Yaskawa INFORM job: X2_38-47,64(1)(90,180).JBI

/JOB
//NAME X2_38-47,64(1)(90,180)
//POS
///NPOS 755,755,755,26,0,0
///TOOL 0
///POSTYPE PULSE
///PULSE
C00000=-10776,-116726,-133110,1428,79202,268
C00001=-121301,-101656,-130574,-15140,106953,-26685
C00002=-120740,-100574,-124017,-14929,103680,-26084
C00003=-120691,-100743,-123189,-14892,103111,-25997
C00004=-120691,-101012,-123023,-14875,102879,-25968
C00005=-120694,-100727,-123199,-14892,103125,-25999
C00006=-120263,-93974,-120700,-15099,105066,-26103
C00007=-120694,-100727,-123199,-14892,103125,-25999
C00008=-121303,-103883,-129892,-15002,105440,-26491
C00009=-121309,-101301,-130428,-15148,107041,-26699
C00010=-120755,-99767,-124232,-14968,104207,-26155
C00011=-120700,-99774,-123449,-14938,103747,-26079
C00012=-120700,-100712,-122892,-14879,102948,-25979
C00013=-120685,-100384,-123078,-14901,103225,-26009
C00014=-120255,-93653,-120581,-15108,105156,-26112
C00015=-120685,-100384,-123078,-14901,103225,-26009
C00016=-121293,-103472,-129753,-15014,105563,-26504
C00017=-114791,-117911,-130965,-19588,74628,-29967
C00018=-114769,-122713,-124135,-20312,68344,-28880
C00019=-114477,-110584,-116158,-20272,69659,-29005
C00020=-114421,-108517,-114081,-20323,69469,-28951
C00021=-114421,-108669,-113508,-20377,69064,-28879
C00022=-114502,-108614,-114130,-20291,69431,-28974
C00023=-116741,-105993,-113204,-19215,69642,-29832
C00024=-114502,-108614,-114130,-20291,69431,-28974
C00025=-119599,-132627,-121815,-19129,61042,-29452
C00026=-135151,-106131,-113172,-10502,66286,-36044
C00027=-134382,-104032,-112419,-10838,66989,-35834
C00028=-133562,-101757,-111587,-11194,67742,-35614
C00029=-135151,-106131,-113172,-10502,66286,-36044
C00030=-114538,-130880,-126635,-20790,65904,-28347
C00031=-100256,-119338,-132400,-19781,92736,17009
C00032=-115252,-134637,-128783,-15911,82002,19716
C00033=-118597,-124593,-122817,-15129,82811,18454
C00034=-119849,-120977,-120499,-14834,83003,18000
C00035=-119848,-121103,-118880,-14863,81976,18124
C00036=-119849,-120977,-120499,-14834,83003,18000
C00037=-134184,-142802,-124917,-2858,68148,11180
C00038=-133176,-135816,-122960,-3144,70568,11480
C00039=-134184,-142802,-124917,-2858,68148,11180
C00040=-110326,-92448,-108322,-23569,98205,21456
C00041=-112623,-92143,-108201,-23254,97666,20755
C00042=-110326,-92448,-108322,-23569,98205,21456
C00043=-105090,-96290,-113946,-24376,100996,22735
C00044=-105112,-88407,-119445,-25319,107768,21250
C00045=-126458,-130213,-127441,18734,86324,-24062
C00046=-122565,-122494,-122126,18005,86127,-22734
C00047=-121090,-119592,-120022,17718,85999,-22241
C00048=-121089,-119765,-118419,17734,84972,-22390
C00049=-121090,-119592,-120022,17718,85999,-22241
C00050=-121090,-119716,-118696,17731,85160,-22363
C00051=-120619,-113401,-116618,17615,86937,-21943
C00052=-121090,-119716,-118696,17731,85160,-22363
C00053=-120691,-116357,-117549,17638,86049,-22096
C00054=-118089,-117386,-117887,17123,85200,-21315
C00055=-120691,-116357,-117549,17638,86049,-22096
C00056=-125936,-126318,-124843,18636,86589,-23840
C00057=-125953,-122568,-132013,18690,92614,-22924
C00058=-117644,-124381,-130105,-6983,115370,67992
C00059=-119593,-136528,-130318,-6950,109138,67660
C00060=-120425,-140611,-129416,-6959,106433,67520
C00061=-120425,-140322,-128375,-6938,105944,67549
C00062=-120287,-139878,-129033,-6943,106584,67561
C00063=-121808,-147552,-131144,-7070,103828,67181
C00064=-120287,-139878,-129033,-6943,106584,67561
C00065=-117523,-124132,-129146,-6933,114921,68065
C00066=-117634,-108923,-132591,-7489,118176,67765
C00067=-119077,-97405,-129626,-2848,111310,9091
C00068=-112934,-122170,-124968,-9693,82630,11419
C00069=-114889,-112052,-118675,-9157,83718,10686
C00070=-115614,-108714,-115508,-8968,83408,10468
C00071=-115614,-108962,-114752,-8976,82823,10510
C00072=-115614,-108688,-115602,-8966,83479,10463
C00073=-130338,-117040,-117457,5173,77211,4432
C00074=-129550,-114521,-116623,4914,77941,4728
C00075=-131152,-119600,-118288,5441,76463,4123
C00076=-115450,-106601,-114144,-9007,83670,10503
C00077=-117654,-103921,-113183,-8408,84218,9737
C00078=-115450,-106601,-114144,-9007,83670,10503
C00079=-112794,-119726,-122752,-9732,82540,11472
C00080=-112816,-114614,-129461,-9677,89201,10949
C00081=-124267,-125778,-125536,12618,81617,-14637
C00082=-121749,-115664,-119377,11934,82621,-13684
C00083=-120813,-112238,-116231,11692,82317,-13397
C00084=-120812,-112414,-115451,11705,81758,-13450
C00085=-120848,-112349,-116241,11703,82272,-13413
C00086=-119586,-107060,-114409,11339,83657,-12862
C00087=-120848,-112349,-116241,11703,82272,-13413
C00088=-124307,-126037,-124767,12644,81031,-14711
C00089=-124281,-122814,-131176,12539,86499,-14147
C00090=-130647,-155525,-127944,40400,54320,-55258
C00091=-124412,-146323,-123540,36852,53123,-52512
C00092=-122059,-142698,-121760,35413,52755,-51453
C00093=-119008,-142706,-121763,33902,51510,-50382
C00094=-122059,-142698,-121760,35413,52755,-51453
C00095=-119813,-142714,-121776,34308,51836,-50667
C00096=-119829,-137326,-119074,33845,52767,-50322
C00097=-119813,-142714,-121776,34308,51836,-50667
C00098=-119893,-119020,-120433,30427,61542,-47434
C00099=-120958,-113296,-116932,30756,62602,-47571
C00100=-120971,-118070,-117370,31352,60722,-48150
C00101=-120958,-113296,-116932,30756,62602,-47571
C00102=-130647,-155525,-127944,40400,54320,-55258
C00103=-121972,-140000,-127461,3525,22047,-40740
C00104=-114503,-126631,-127045,-28228,88345,-28238
C00105=-115418,-120062,-121213,-28067,87856,-28460
C00106=-115767,-117777,-118144,-28010,87108,-28410
C00107=-115767,-117863,-117333,-28016,86625,-28294
C00108=-115798,-117876,-117463,-28010,86680,-28319
C00109=-115506,-111666,-115391,-28051,88476,-28642
C00110=-115798,-117876,-117463,-28010,86680,-28319
C00111=-114535,-126949,-125608,-28226,87406,-28022
C00112=-81132,-132100,-132064,-22325,96940,-18748
C00113=-82014,-125321,-126186,-22252,96583,-18997
C00114=-82351,-123063,-123074,-22185,95795,-18971
C00115=-82354,-123167,-122323,-22159,95314,-18883
C00116=-82329,-123147,-122467,-22165,95412,-18892
C00117=-83163,-116500,-120334,-22218,97147,-19515
C00118=-82329,-123147,-122467,-22165,95412,-18892
C00119=-81992,-125617,-124767,-22197,95637,-18813
C00120=-81110,-132470,-130662,-22266,95968,-18558
C00121=-88413,-113418,-132573,-32131,117765,-52556
C00122=-88284,-148255,-125485,-32887,110398,-70729
C00123=-90408,-157751,-124889,-32381,105124,-70012
C00124=-91344,-160468,-123864,-32301,103041,-69779
C00125=-91347,-158891,-122215,-32272,102866,-69728
C00126=-106792,-136481,-118062,-29763,111204,-74713
C00127=-106248,-142899,-119829,-29161,109458,-74003
C00128=-106792,-136481,-118062,-29763,111204,-74713
C00129=-72811,-175927,-123443,-35029,98716,-64074
C00130=-76149,-179694,-124176,-35896,96158,-64586
C00131=-72811,-175927,-123443,-35029,98716,-64074
C00132=-69241,-166504,-125806,-34856,105362,-64752
C00133=-100814,-129767,-126176,-13403,120642,-68982
C00134=-124653,-147507,-132240,11278,113041,-68250
C00135=-122082,-159833,-132453,11465,106593,-67927
C00136=-120959,-163108,-131284,11603,104077,-67764
C00137=-120958,-161905,-130051,11594,103939,-67777
C00138=-120958,-161991,-130311,11601,104052,-67766
C00139=-120981,-170969,-132443,11421,100817,-68083
C00140=-120958,-161991,-130311,11601,104052,-67766
C00141=-120973,-170778,-133362,11455,101467,-68019
C00142=-117530,-170630,-133328,12326,101017,-66845
C00143=-120973,-170778,-133362,11455,101467,-68019
C00144=-124784,-154865,-133680,10989,110216,-68576
C00145=-122322,-137878,-131274,-5971,121779,-67906
C00146=-120548,-145044,-127252,-18536,119036,-66813
C00147=-120555,-156847,-127343,-17506,113306,-65855
C00148=-120558,-160498,-126573,-17182,111059,-65507
C00149=-120558,-158961,-124938,-17154,110851,-65476
C00150=-120618,-159187,-125406,-17199,111003,-65522
C00151=-120626,-166810,-127194,-16864,108302,-65121
C00152=-120618,-159187,-125406,-17199,111003,-65522
C00153=-120603,-144021,-125705,-18473,118618,-66761
C00154=-115387,-132374,-123926,-32562,106734,-81694
C00155=-118372,-141379,-123449,-32107,101406,-81342
C00156=-119656,-144207,-122551,-32012,99204,-81226
C00157=-119656,-143343,-121080,-31963,98811,-81114
C00158=-119656,-144508,-123075,-32029,99348,-81268
C00159=-131320,-114613,-113969,-28597,111497,-86004
C00160=-131699,-120616,-115930,-28265,109708,-85685
C00161=-131320,-114613,-113969,-28597,111497,-86004
C00162=-105239,-169544,-124716,-37289,88926,-74807
C00163=-108884,-170779,-124983,-37802,86985,-75650
C00164=-105239,-169544,-124716,-37289,88926,-74807
C00165=-99694,-161827,-127351,-36723,95805,-74832
C00166=-131992,-100814,-126478,-21663,116809,46067
C00167=-134007,-144842,-130967,-18968,105768,42043
C00168=-134012,-143545,-127522,-18820,104388,42265
C00169=-134287,-143929,-127856,-18860,104334,42172
C00170=-133739,-135079,-123901,-19000,106464,42030
C00171=-134287,-143184,-126185,-18799,103720,42271
C00172=-134064,-144330,-127677,-2767,111202,58459
C00173=-134007,-143438,-127424,-2760,111507,58474
C00174=-135126,-137550,-119428,14300,119099,83463
C00175=-134030,-140788,-121209,15013,118595,84384
C00176=-134030,-142235,-124150,15187,119626,84533
C00177=-119630,-122416,-133334,16028,118546,61096
C00178=-134341,-125466,-134740,10815,104436,21672
C00179=-120614,-100166,-121253,7350,89365,-11707
C00180=-120622,-93660,-109595,7359,85566,-11930
C00181=-122164,-90812,-108950,7802,86761,-12352
C00182=-122198,-95853,-109304,7828,84412,-12509
C00183=-122164,-91688,-107664,7808,85529,-12428
C00184=-120622,-94101,-108793,7365,84850,-11972
C00185=-122951,-73862,-99576,-7929,88190,4985
C00186=-120621,-96600,-101892,-16342,67221,11741
C00187=-120621,-96191,-103793,-16192,68548,11553
C00188=-120639,-92247,-111396,-15618,75005,10677
C00189=-188010,-107595,-125638,17104,94805,-24250
C00190=-188020,-110122,-123495,17031,92300,-24603
C00191=-187252,-116827,-124472,16830,89421,-24740
C00192=-188438,-109992,-122083,17102,91614,-24840
C00193=-188123,-110345,-123595,17051,92269,-24642
C00194=-188114,-107825,-125741,17124,94773,-24289
C00195=-177438,-122732,-133224,14695,89877,-21402
C00196=-133569,-113989,-134534,14289,94663,-20149
C00197=-119624,-110386,-135117,7911,77851,-79525
C00198=-120615,-106635,-127104,8473,74968,-80030
C00199=-127138,-106639,-125023,15586,75013,-81251
C00200=-130661,-111022,-125418,19776,73192,-82197
C00201=-120615,-106612,-127117,8473,74988,-80029
C00202=-122620,-125184,-116655,35316,53565,-49443
C00203=-120598,-121294,-114839,33833,53482,-48472
C00204=-120551,-127900,-115071,35213,50759,-49502
C00205=-120377,-147941,-114075,41532,42004,-53628
C00206=-120733,-119186,-113678,30224,65857,-57863
C00207=-122683,-120749,-115245,30946,66698,-58435
C00208=-127694,-124296,-119025,32687,68997,-59841
C00209=-127721,-118762,-131765,31151,78153,-27047
C00210=-126237,-112945,-130032,468,65797,-4909
C00211=-102361,-117345,-122757,-6013,83638,2551
C00212=-102141,-118134,-119975,-6094,81548,2725
C00213=-99061,-100059,-114136,-7526,92006,6303
C00214=-118448,-105217,-116092,-2994,89929,-3052
C00215=-122253,-105715,-115580,-4099,87909,4316
C00216=-120609,-124185,-121101,-4570,77097,5239
C00217=-120610,-123821,-123927,-4542,79018,5168
C00218=-108948,-109237,-131335,-7817,91844,8301
C00219=-115305,-101104,-129841,-7326,117578,44729
C00220=-120606,-132359,-125648,-5649,119733,79611
C00221=-120606,-131978,-122596,-5547,118059,79698
C00222=-120699,-131888,-121364,-5538,117345,79699
C00223=-120606,-132064,-121373,-5500,117266,79739
C00224=-120607,-132636,-121567,-5491,117090,79751
C00225=-120606,-132150,-119920,-13765,116589,67538
C00226=-120606,-131851,-120987,-13891,117375,67436
C00227=-120606,-132395,-123921,-14113,118858,67242
C00228=-111305,-120759,-132293,-17375,98141,32748
C00229=-120609,-124691,-119154,-16638,71592,14867
C00230=-120609,-124440,-116582,-16774,70197,15066
C00231=-120609,-124277,-115533,-16830,69659,15144
C00232=-120609,-125082,-119997,8806,76841,-5950
C00233=-120609,-124819,-119897,8803,76914,-5945
C00234=-120609,-124768,-117835,18246,76542,-19045
C00235=-120609,-124884,-118955,18205,77141,-18954
C00236=-120609,-124961,-121688,18108,78705,-18718
C00237=-132640,-106780,-128323,23054,110263,28369
C00238=-120602,-139315,-124713,24306,112781,84362
C00239=-120602,-138068,-121544,24057,111582,84094
C00240=-120602,-137520,-120260,23964,111115,83992
C00241=-111171,-137450,-123178,3338,116163,79197
C00242=-120602,-139000,-123563,90,115805,75571
C00243=-109330,-134151,-116420,-27663,112170,68648
C00244=-107669,-134044,-117364,-27346,113285,69054
C00245=-103576,-133216,-119553,-26575,116197,70036
C00246=-103610,-135048,-130246,-28186,121222,68648
C00247=-111190,-129681,-128447,-36946,96833,72948
C00248=-111854,-129032,-128166,-43025,93670,81713
C00249=-147502,-118658,-119533,-35927,77679,72524
C00250=-147511,-119004,-116560,-36172,76036,73070
C00251=-147515,-119022,-115332,-36276,75411,73279
C00252=-147547,-116234,-125968,-15022,114340,70681
C00253=-147515,-116012,-125840,-15022,114380,70688
C00254=-147502,-115929,-125780,-17177,108602,60467
C00255=-147494,-115895,-125723,-16722,102508,50684
C00256=-147493,-115916,-125679,-13964,96968,41110
C00257=-147497,-115970,-125656,-10645,93613,33926
C00258=-147501,-116025,-125648,-8199,92025,29507
C00259=-147506,-116072,-125646,-5516,90867,25066
C00260=-147508,-116095,-125646,-5516,90856,25066
C00261=-147505,-115163,-126691,-5523,91973,25018
C00262=-147498,-112805,-128627,-5545,94366,24915
C00263=-120610,-124729,-127429,5691,77135,-5542
C00264=-120610,-125478,-124917,5733,75213,-5631
C00265=-93224,-108496,-118221,-17160,84932,17314
C00266=-100404,-109639,-120638,-9099,85725,5885
C00267=-100577,-112155,-122052,-6607,85486,-528
C00268=-115338,-131033,-127093,4056,76541,-4536
C00269=-121145,-125062,-125115,1467,77680,-1578
C00270=-113474,-126239,-125199,-4571,76718,-3065
C00271=-116327,-126679,-125338,-2161,76267,-5597
C00272=-113490,-126055,-125151,-4559,76778,-3077
C00273=-117667,-122970,-124192,-3214,77575,-4511
C00274=-120712,-121109,-123606,-2232,78069,-5542
C00275=-125774,-129632,-127388,3161,76112,-11172
C00276=-120611,-124694,-128184,1477,78993,-9385
C00277=2000,-120083,-131752,1890,40973,0
C00278=-10776,-116726,-133110,1428,79202,268
C00279=-121301,-101656,-130574,-15140,106953,-26685
C00280=-120740,-100574,-124017,-14929,103680,-26084
C00281=-120691,-100743,-123189,-14892,103111,-25997
C00282=-120691,-101012,-123023,-14875,102879,-25968
C00283=-120694,-100727,-123199,-14892,103125,-25999
C00284=-120263,-93974,-120700,-15099,105066,-26103
C00285=-120694,-100727,-123199,-14892,103125,-25999
C00286=-121303,-103883,-129892,-15002,105440,-26491
C00287=-121309,-101301,-130428,-15148,107041,-26699
C00288=-120755,-99767,-124232,-14968,104207,-26155
C00289=-120700,-99774,-123449,-14938,103747,-26079
C00290=-120700,-100712,-122892,-14879,102948,-25979
C00291=-120685,-100384,-123078,-14901,103225,-26009
C00292=-120255,-93653,-120581,-15108,105156,-26112
C00293=-120685,-100384,-123078,-14901,103225,-26009
C00294=-121293,-103472,-129753,-15014,105563,-26504
C00295=-114791,-117911,-130965,-19588,74628,-29967
C00296=-114769,-122713,-124135,-20312,68344,-28880
C00297=-114477,-110584,-116158,-20272,69659,-29005
C00298=-114421,-108517,-114081,-20323,69469,-28951
C00299=-114421,-108669,-113508,-20377,69064,-28879
C00300=-114502,-108614,-114130,-20291,69431,-28974
C00301=-116741,-105993,-113204,-19215,69642,-29832
C00302=-114502,-108614,-114130,-20291,69431,-28974
C00303=-119599,-132627,-121815,-19129,61042,-29452
C00304=-135151,-106131,-113172,-10502,66286,-36044
C00305=-134382,-104032,-112419,-10838,66989,-35834
C00306=-133562,-101757,-111587,-11194,67742,-35614
C00307=-135151,-106131,-113172,-10502,66286,-36044
C00308=-114538,-130880,-126635,-20790,65904,-28347
C00309=-100256,-119338,-132400,-19781,92736,17009
C00310=-115252,-134637,-128783,-15911,82002,19716
C00311=-118597,-124593,-122817,-15129,82811,18454
C00312=-119849,-120977,-120499,-14834,83003,18000
C00313=-119848,-121103,-118880,-14863,81976,18124
C00314=-119849,-120977,-120499,-14834,83003,18000
C00315=-134184,-142802,-124917,-2858,68148,11180
C00316=-133176,-135816,-122960,-3144,70568,11480
C00317=-134184,-142802,-124917,-2858,68148,11180
C00318=-110326,-92448,-108322,-23569,98205,21456
C00319=-112623,-92143,-108201,-23254,97666,20755
C00320=-110326,-92448,-108322,-23569,98205,21456
C00321=-105090,-96290,-113946,-24376,100996,22735
C00322=-105112,-88407,-119445,-25319,107768,21250
C00323=-126458,-130213,-127441,18734,86324,-24062
C00324=-122565,-122494,-122126,18005,86127,-22734
C00325=-121090,-119592,-120022,17718,85999,-22241
C00326=-121089,-119765,-118419,17734,84972,-22390
C00327=-121090,-119592,-120022,17718,85999,-22241
C00328=-121090,-119716,-118696,17731,85160,-22363
C00329=-120619,-113401,-116618,17615,86937,-21943
C00330=-121090,-119716,-118696,17731,85160,-22363
C00331=-120691,-116357,-117549,17638,86049,-22096
C00332=-118089,-117386,-117887,17123,85200,-21315
C00333=-120691,-116357,-117549,17638,86049,-22096
C00334=-125936,-126318,-124843,18636,86589,-23840
C00335=-125953,-122568,-132013,18690,92614,-22924
C00336=-117644,-124381,-130105,-6983,115370,67992
C00337=-119593,-136528,-130318,-6950,109138,67660
C00338=-120425,-140611,-129416,-6959,106433,67520
C00339=-120425,-140322,-128375,-6938,105944,67549
C00340=-120287,-139878,-129033,-6943,106584,67561
C00341=-121808,-147552,-131144,-7070,103828,67181
C00342=-120287,-139878,-129033,-6943,106584,67561
C00343=-117523,-124132,-129146,-6933,114921,68065
C00344=-117634,-108923,-132591,-7489,118176,67765
C00345=-119077,-97405,-129626,-2848,111310,9091
C00346=-112934,-122170,-124968,-9693,82630,11419
C00347=-114889,-112052,-118675,-9157,83718,10686
C00348=-115614,-108714,-115508,-8968,83408,10468
C00349=-115614,-108962,-114752,-8976,82823,10510
C00350=-115614,-108688,-115602,-8966,83479,10463
C00351=-130338,-117040,-117457,5173,77211,4432
C00352=-129550,-114521,-116623,4914,77941,4728
C00353=-131152,-119600,-118288,5441,76463,4123
C00354=-115450,-106601,-114144,-9007,83670,10503
C00355=-117654,-103921,-113183,-8408,84218,9737
C00356=-115450,-106601,-114144,-9007,83670,10503
C00357=-112794,-119726,-122752,-9732,82540,11472
C00358=-112816,-114614,-129461,-9677,89201,10949
C00359=-124267,-125778,-125536,12618,81617,-14637
C00360=-121749,-115664,-119377,11934,82621,-13684
C00361=-120813,-112238,-116231,11692,82317,-13397
C00362=-120812,-112414,-115451,11705,81758,-13450
C00363=-120848,-112349,-116241,11703,82272,-13413
C00364=-119586,-107060,-114409,11339,83657,-12862
C00365=-120848,-112349,-116241,11703,82272,-13413
C00366=-124307,-126037,-124767,12644,81031,-14711
C00367=-124281,-122814,-131176,12539,86499,-14147
C00368=-130647,-155525,-127944,40400,54320,-55258
C00369=-124412,-146323,-123540,36852,53123,-52512
C00370=-122059,-142698,-121760,35413,52755,-51453
C00371=-119008,-142706,-121763,33902,51510,-50382
C00372=-122059,-142698,-121760,35413,52755,-51453
C00373=-119813,-142714,-121776,34308,51836,-50667
C00374=-119829,-137326,-119074,33845,52767,-50322
C00375=-119813,-142714,-121776,34308,51836,-50667
C00376=-119893,-119020,-120433,30427,61542,-47434
C00377=-120958,-113296,-116932,30756,62602,-47571
C00378=-120971,-118070,-117370,31352,60722,-48150
C00379=-120958,-113296,-116932,30756,62602,-47571
C00380=-130647,-155525,-127944,40400,54320,-55258
C00381=-121972,-140000,-127461,3525,22047,-40740
C00382=-114503,-126631,-127045,-28228,88345,-28238
C00383=-115418,-120062,-121213,-28067,87856,-28460
C00384=-115767,-117777,-118144,-28010,87108,-28410
C00385=-115767,-117863,-117333,-28016,86625,-28294
C00386=-115798,-117876,-117463,-28010,86680,-28319
C00387=-115506,-111666,-115391,-28051,88476,-28642
C00388=-115798,-117876,-117463,-28010,86680,-28319
C00389=-114535,-126949,-125608,-28226,87406,-28022
C00390=-81132,-132100,-132064,-22325,96940,-18748
C00391=-82014,-125321,-126186,-22252,96583,-18997
C00392=-82351,-123063,-123074,-22185,95795,-18971
C00393=-82354,-123167,-122323,-22159,95314,-18883
C00394=-82329,-123147,-122467,-22165,95412,-18892
C00395=-83163,-116500,-120334,-22218,97147,-19515
C00396=-82329,-123147,-122467,-22165,95412,-18892
C00397=-81992,-125617,-124767,-22197,95637,-18813
C00398=-81110,-132470,-130662,-22266,95968,-18558
C00399=-88413,-113418,-132573,-32131,117765,-52556
C00400=-88284,-148255,-125485,-32887,110398,-70729
C00401=-90408,-157751,-124889,-32381,105124,-70012
C00402=-91344,-160468,-123864,-32301,103041,-69779
C00403=-91347,-158891,-122215,-32272,102866,-69728
C00404=-106792,-136481,-118062,-29763,111204,-74713
C00405=-106248,-142899,-119829,-29161,109458,-74003
C00406=-106792,-136481,-118062,-29763,111204,-74713
C00407=-72811,-175927,-123443,-35029,98716,-64074
C00408=-76149,-179694,-124176,-35896,96158,-64586
C00409=-72811,-175927,-123443,-35029,98716,-64074
C00410=-69241,-166504,-125806,-34856,105362,-64752
C00411=-100814,-129767,-126176,-13403,120642,-68982
C00412=-124653,-147507,-132240,11278,113041,-68250
C00413=-122082,-159833,-132453,11465,106593,-67927
C00414=-120959,-163108,-131284,11603,104077,-67764
C00415=-120958,-161905,-130051,11594,103939,-67777
C00416=-120958,-161991,-130311,11601,104052,-67766
C00417=-120981,-170969,-132443,11421,100817,-68083
C00418=-120958,-161991,-130311,11601,104052,-67766
C00419=-120973,-170778,-133362,11455,101467,-68019
C00420=-117530,-170630,-133328,12326,101017,-66845
C00421=-120973,-170778,-133362,11455,101467,-68019
C00422=-124784,-154865,-133680,10989,110216,-68576
C00423=-122322,-137878,-131274,-5971,121779,-67906
C00424=-120548,-145044,-127252,-18536,119036,-66813
C00425=-120555,-156847,-127343,-17506,113306,-65855
C00426=-120558,-160498,-126573,-17182,111059,-65507
C00427=-120558,-158961,-124938,-17154,110851,-65476
C00428=-120618,-159187,-125406,-17199,111003,-65522
C00429=-120626,-166810,-127194,-16864,108302,-65121
C00430=-120618,-159187,-125406,-17199,111003,-65522
C00431=-120603,-144021,-125705,-18473,118618,-66761
C00432=-115387,-132374,-123926,-32562,106734,-81694
C00433=-118372,-141379,-123449,-32107,101406,-81342
C00434=-119656,-144207,-122551,-32012,99204,-81226
C00435=-119656,-143343,-121080,-31963,98811,-81114
C00436=-119656,-144508,-123075,-32029,99348,-81268
C00437=-131320,-114613,-113969,-28597,111497,-86004
C00438=-131699,-120616,-115930,-28265,109708,-85685
C00439=-131320,-114613,-113969,-28597,111497,-86004
C00440=-105239,-169544,-124716,-37289,88926,-74807
C00441=-108884,-170779,-124983,-37802,86985,-75650
C00442=-105239,-169544,-124716,-37289,88926,-74807
C00443=-99694,-161827,-127351,-36723,95805,-74832
C00444=-131992,-100814,-126478,-21663,116809,46067
C00445=-134007,-144842,-130967,-18968,105768,42043
C00446=-134012,-143545,-127522,-18820,104388,42265
C00447=-134287,-143929,-127856,-18860,104334,42172
C00448=-133739,-135079,-123901,-19000,106464,42030
C00449=-134287,-143184,-126185,-18799,103720,42271
C00450=-134064,-144330,-127677,-2767,111202,58459
C00451=-134007,-143438,-127424,-2760,111507,58474
C00452=-135126,-137550,-119428,14300,119099,83463
C00453=-134030,-140788,-121209,15013,118595,84384
C00454=-134030,-142235,-124150,15187,119626,84533
C00455=-119630,-122416,-133334,16028,118546,61096
C00456=-134341,-125466,-134740,10815,104436,21672
C00457=-120614,-100166,-121253,7350,89365,-11707
C00458=-120622,-93660,-109595,7359,85566,-11930
C00459=-122164,-90812,-108950,7802,86761,-12352
C00460=-122198,-95853,-109304,7828,84412,-12509
C00461=-122164,-91688,-107664,7808,85529,-12428
C00462=-120622,-94101,-108793,7365,84850,-11972
C00463=-122951,-73862,-99576,-7929,88190,4985
C00464=-120621,-96600,-101892,-16342,67221,11741
C00465=-120621,-96191,-103793,-16192,68548,11553
C00466=-120639,-92247,-111396,-15618,75005,10677
C00467=-188010,-107595,-125638,17104,94805,-24250
C00468=-188020,-110122,-123495,17031,92300,-24603
C00469=-187252,-116827,-124472,16830,89421,-24740
C00470=-188438,-109992,-122083,17102,91614,-24840
C00471=-188123,-110345,-123595,17051,92269,-24642
C00472=-188114,-107825,-125741,17124,94773,-24289
C00473=-177438,-122732,-133224,14695,89877,-21402
C00474=-133569,-113989,-134534,14289,94663,-20149
C00475=-119624,-110386,-135117,7911,77851,-79525
C00476=-120615,-106635,-127104,8473,74968,-80030
C00477=-127138,-106639,-125023,15586,75013,-81251
C00478=-130661,-111022,-125418,19776,73192,-82197
C00479=-120615,-106612,-127117,8473,74988,-80029
C00480=-122620,-125184,-116655,35316,53565,-49443
C00481=-120598,-121294,-114839,33833,53482,-48472
C00482=-120551,-127900,-115071,35213,50759,-49502
C00483=-120377,-147941,-114075,41532,42004,-53628
C00484=-120733,-119186,-113678,30224,65857,-57863
C00485=-122683,-120749,-115245,30946,66698,-58435
C00486=-127694,-124296,-119025,32687,68997,-59841
C00487=-127721,-118762,-131765,31151,78153,-27047
C00488=-126237,-112945,-130032,468,65797,-4909
C00489=-102361,-117345,-122757,-6013,83638,2551
C00490=-102141,-118134,-119975,-6094,81548,2725
C00491=-99061,-100059,-114136,-7526,92006,6303
C00492=-118448,-105217,-116092,-2994,89929,-3052
C00493=-122253,-105715,-115580,-4099,87909,4316
C00494=-120609,-124185,-121101,-4570,77097,5239
C00495=-120610,-123821,-123927,-4542,79018,5168
C00496=-108948,-109237,-131335,-7817,91844,8301
C00497=-115305,-101104,-129841,-7326,117578,44729
C00498=-120606,-132359,-125648,-5649,119733,79611
C00499=-120606,-131978,-122596,-5547,118059,79698
C00500=-120699,-131888,-121364,-5538,117345,79699
C00501=-120606,-132064,-121373,-5500,117266,79739
C00502=-120606,-131696,-121291,-5509,117403,79735
C00503=-120606,-131546,-119742,-13806,116783,67512
C00504=-120606,-131851,-120987,-13891,117375,67436
C00505=-120606,-132395,-123921,-14113,118858,67242
C00506=-111305,-120759,-132293,-17375,98141,32748
C00507=-120609,-124691,-119154,-16638,71592,14867
C00508=-120609,-124440,-116582,-16774,70197,15066
C00509=-120609,-124277,-115533,-16830,69659,15144
C00510=-120609,-125082,-119997,8806,76841,-5950
C00511=-120609,-124819,-119897,8803,76914,-5945
C00512=-120609,-124768,-117835,18246,76542,-19045
C00513=-120609,-124884,-118955,18205,77141,-18954
C00514=-120609,-124961,-121688,18108,78705,-18718
C00515=-132640,-106780,-128323,23054,110263,28369
C00516=-120602,-139315,-124713,24306,112781,84362
C00517=-120602,-138068,-121544,24057,111582,84094
C00518=-120602,-137520,-120260,23964,111115,83992
C00519=-111171,-137450,-123178,3338,116163,79197
C00520=-120602,-139000,-123563,90,115805,75571
C00521=-109330,-134151,-116420,-27663,112170,68648
C00522=-107669,-134044,-117364,-27346,113285,69054
C00523=-103576,-133216,-119553,-26575,116197,70036
C00524=-103610,-135048,-130246,-28186,121222,68648
C00525=-111190,-129681,-128447,-36946,96833,72948
C00526=-111854,-129032,-128166,-43025,93670,81713
C00527=-147502,-118658,-119533,-35927,77679,72524
C00528=-147511,-119004,-116560,-36172,76036,73070
C00529=-147515,-119022,-115332,-36276,75411,73279
C00530=-147547,-116234,-125968,-15022,114340,70681
C00531=-147515,-116012,-125840,-15022,114380,70688
C00532=-147502,-115929,-125780,-17177,108602,60467
C00533=-147494,-115895,-125723,-16722,102508,50684
C00534=-147493,-115916,-125679,-13964,96968,41110
C00535=-147497,-115970,-125656,-10645,93613,33926
C00536=-147501,-116025,-125648,-8199,92025,29507
C00537=-147506,-116072,-125646,-5516,90867,25066
C00538=-147508,-116095,-125646,-5516,90856,25066
C00539=-147505,-115163,-126691,-5523,91973,25018
C00540=-147498,-112805,-128627,-5545,94366,24915
C00541=-120610,-124729,-127429,5691,77135,-5542
C00542=-120610,-125478,-124917,5733,75213,-5631
C00543=-121145,-125062,-125115,1467,77680,-1578
C00544=-93224,-108496,-118221,-17160,84932,17314
C00545=-100404,-109639,-120638,-9099,85725,5885
C00546=-100577,-112155,-122052,-6607,85486,-528
C00547=-115338,-131033,-127093,4056,76541,-4536
C00548=-121145,-125062,-125115,1467,77680,-1578
C00549=-113474,-126239,-125199,-4571,76718,-3065
C00550=-116327,-126679,-125338,-2161,76267,-5597
C00551=-113490,-126055,-125151,-4559,76778,-3077
C00552=-117667,-122970,-124192,-3214,77575,-4511
C00553=-120712,-121109,-123606,-2232,78069,-5542
C00554=-125774,-129632,-127388,3161,76112,-11172
C00555=-120611,-124694,-128184,1477,78993,-9385
C00556=2000,-120083,-131752,1890,40973,0
C00557=-15972,-110889,-128286,-10965,59905,-43045
C00558=-101389,-60822,-75148,6919,68546,-70102
C00559=-115790,69230,64798,-8053,66131,-71909
C00560=-120830,71540,61874,-4756,55589,-66514
C00561=-120535,76858,72419,-5134,51864,-66212
C00562=-120418,79487,77321,-5314,50212,-66075
C00563=-120418,81305,81326,-5435,48689,-65991
C00564=-120418,79487,77321,-5314,50212,-66075
C00565=-121101,73566,71896,-4942,50464,-66384
C00566=-120640,77942,77238,-5256,49458,-66131
C00567=-121101,73566,71896,-4942,50464,-66384
C00568=-121527,66226,57370,-4418,55590,-66797
C00569=-120817,46858,51705,6808,46216,-80289
C00570=-120487,52530,62238,7041,42645,-80409
C00571=-120357,55197,66992,7170,41090,-80474
C00572=-120357,57219,71131,7393,39594,-80606
C00573=-120357,55197,66992,7170,41090,-80474
C00574=-121171,51687,64922,7778,40638,-80922
C00575=-120657,55397,69123,7546,39918,-80729
C00576=-121171,51687,64922,7778,40638,-80922
C00577=-121648,43436,49847,7373,45678,-80715
C00578=-109578,66950,51259,-9202,73878,-70224
C00579=-101389,-60822,-75148,6919,68546,-70102
C00580=-96929,-90691,-89138,5080,61517,-23019
C00581=-96929,-90691,-89138,5080,61517,27168
C00582=-133997,38575,-5386,4879,105902,64390
C00583=-134430,35731,-4221,4855,103756,64161
C00584=-134605,34491,-3252,4839,102536,64054
C00585=-134604,34193,-2477,4825,101908,64030
C00586=-134605,34666,-3678,4847,102887,64068
C00587=-133324,38381,1851,4717,101326,64430
C00588=-133984,36157,-436,4773,101627,64224
C00589=-133324,38381,1851,4717,101326,64430
C00590=-132740,42105,45,4739,104308,64739
C00591=-134038,40743,-3018,12196,109842,66951
C00592=-134155,37294,-2552,12029,107844,66703
C00593=-134138,36860,-901,11936,106627,66584
C00594=-134138,36533,-42,11887,105945,66515
C00595=-134138,36618,-275,11900,106128,66533
C00596=-134308,36004,-906,11910,106222,66482
C00597=-134138,36772,-681,11923,106449,66566
C00598=-133552,41863,-495,12102,108819,67011
C00599=-143157,-5596,-33734,3459,84138,-17748
C00600=-146617,-6443,-23161,4534,77380,-19112
C00601=-149281,-2495,-17370,9500,77350,-25048
C00602=-149281,-2461,-16373,9521,76762,-25094
C00603=-149281,-2503,-17669,9494,77528,-25035
C00604=-148457,-726,-16200,9269,77441,-24757
C00605=-149281,-2503,-17669,9494,77528,-25035
C00606=-157589,4412,-9593,22718,80450,-41052
C00607=-157226,5016,-8132,22675,79802,-41042
C00608=-156592,4240,-8798,22542,79640,-40841
C00609=-157226,4947,-9136,22642,80340,-40940
C00610=-149281,-2387,-22338,9412,80423,-24814
C00611=-159526,23962,790,32225,80504,55500
C00612=-158922,24925,5721,32299,78113,55050
C00613=-158682,25458,8512,32395,76792,54763
C00614=-158681,25549,9587,32465,76269,54609
C00615=-159783,23528,6240,32612,77557,54544
C00616=-160104,22984,7189,32780,76948,54233
C00617=-159169,24509,8648,32575,76492,54477
C00618=-160104,22984,7189,32780,76948,54233
C00619=-160967,21427,101,32642,80299,54873
C00620=-147551,27169,-6215,28445,81493,60312
C00621=-147017,27605,-1759,28452,79091,59917
C00622=-146805,27832,419,28491,77938,59710
C00623=-146803,27699,1600,28565,77235,59535
C00624=-147749,25558,-2150,28746,78615,59523
C00625=-148390,24338,-1607,29025,77984,59121
C00626=-147556,26192,183,28786,77573,59333
C00627=-148390,24338,-1607,29025,77984,59121
C00628=-149162,23542,-7999,28991,81344,59682
C00629=-148025,26294,-7040,28591,81698,60189
C00630=-147485,26714,-2602,28593,79299,59793
C00631=-147271,26975,-740,28610,78335,59633
C00632=-147270,26798,747,28702,77445,59410
C00633=-147271,26975,-740,28610,78335,59633
C00634=-147888,25428,-868,28863,77908,59292
C00635=-147063,27300,949,28626,77494,59501
C00636=-147888,25428,-868,28863,77908,59292
C00637=-148652,24637,-7261,28828,81272,59852
C00638=-129846,-17397,-52274,16165,101048,68229
C00639=-103949,-6271,-30701,7884,96105,76175
C00640=-94102,16895,-5866,4380,94047,79161
C00641=-94024,14878,-3719,4358,91692,79105
C00642=-93993,14152,-2780,4351,90742,79083
C00643=-93993,14253,-1030,4349,89719,79047
C00644=-93993,14152,-2780,4351,90742,79083
C00645=-93685,20015,4382,4321,89334,79138
C00646=-93881,17120,1686,4338,89515,79078
C00647=-93685,20015,4382,4321,89334,79138
C00648=-93796,22544,1176,4343,92603,79213
C00649=-95224,-25687,-42365,27028,60157,72238
C00650=-94111,-23276,-36997,26973,57954,72128
C00651=-93676,-22234,-34203,27071,56755,71994
C00652=-93677,-22196,-33100,27266,56165,71832
C00653=-94095,-27015,-37738,27384,56638,71778
C00654=-94165,-26445,-35973,27662,55954,71554
C00655=-93910,-23559,-33944,27450,56079,71704
C00656=-94165,-26445,-35973,27662,55954,71554
C00657=-95768,-30118,-43626,27714,58991,71694
C00658=-98687,-54699,-75805,10421,73482,70446
C00659=-149776,12587,-27486,12781,89603,-18869
C00660=-147726,21450,-15619,10072,89467,-18633
C00661=-146190,28089,-6729,8043,89366,-18457
C00662=-138712,21584,-10452,-6744,81967,66
C00663=-138085,14099,-20532,-6917,84360,139
C00664=-145864,23955,-12684,8284,88428,-27874
C00665=-146885,25936,-8147,8552,86771,-28313
C00666=-147056,24986,-14909,8600,90423,-28118
C00667=-133623,24371,-15503,-12505,92341,-3955
C00668=-141603,20096,-23343,17631,90771,45924
C00669=-175362,59573,37827,46975,74531,48445
C00670=-174398,62305,44598,47324,72110,47721
C00671=-174360,66018,50115,47663,71067,47209
C00672=-172482,53047,37078,44374,62215,46865
C00673=-172628,50226,32658,43982,63214,47275
C00674=-173442,46522,25111,43389,65629,48000
C00675=-175751,57855,36014,51960,82937,49775
C00676=-174271,55569,37030,51911,80967,49439
C00677=-173860,55550,38133,51931,80301,49277
C00678=-174439,62023,45522,52154,79857,48710
C00679=-175386,75453,61635,55272,87245,48999
C00680=-176596,75085,57687,55306,89275,49600
C00681=-162891,39596,10758,46944,80889,54952
C00682=-161747,40468,15313,46928,78664,54425
C00683=-163273,53880,32001,50799,82657,52192
C00684=-162010,46460,23909,50499,82720,52878
C00685=-160571,34350,9025,46543,78569,54946
C00686=-161741,33529,4546,46578,80799,55455
C00687=-147996,42947,122,12460,106294,61459
C00688=-148226,40262,1426,12324,104193,61162
C00689=-146766,53866,17608,9771,108156,61626
C00690=-145306,48527,11741,9899,108797,62196
C00691=-146773,35404,-3590,12275,104564,61692
C00692=-146547,41093,-8751,12742,110494,62402
C00693=-170472,-48867,-31078,12436,82300,51309
C00694=-161833,-30139,-32162,12294,91042,55174
C00695=-111128,62365,52281,-11955,55160,-64549
C00696=-111043,67239,62048,-12539,51743,-64100
C00697=-108427,49473,54066,-27881,35011,-61543
C00698=-110512,52951,57928,-26501,33808,-62418
C00699=-113115,71610,67239,-11613,50506,-64854
C00700=-113215,66301,56846,-11015,54091,-65302
C00701=-121898,77388,65564,1855,57299,-70150
C00702=-121470,82378,75801,1732,53556,-70040
C00703=-123195,67922,64647,6849,45018,-71451
C00704=-122125,64607,60584,6056,45727,-70899
C00705=-120225,78262,70725,1119,54542,-69513
C00706=-120651,73746,61164,1269,58111,-69644
C00707=-113189,52303,49996,7645,51731,-77534
C00708=-112734,56976,59397,7777,48333,-77603
C00709=-114820,45850,55114,15931,36430,-80431
C00710=-110545,39461,48380,12117,36535,-77984
C00711=-108220,49577,51136,5183,49245,-75539
C00712=-108655,45336,42401,5185,52457,-75559
C00713=-161833,-30139,-32162,12294,91042,55174
C00714=-170472,-47446,-27408,12476,80805,51159
C00715=-92809,-22406,-39596,-2559,87564,76845
C00716=-93205,-23584,-36354,-2491,84954,76766
C00717=-93735,-23855,-34916,-2398,83915,76608
C00718=-94613,-23604,-34737,-2238,83909,76313
C00719=-94250,-23197,-36080,-2300,84954,76417
C00720=-93848,-22027,-39325,-2370,87561,76502
C00721=-94651,-21766,-39138,7100,89212,77956
C00722=-94455,-23170,-36061,7070,86599,77874
C00723=-95157,-23346,-34555,7184,85647,77584
C00724=-93759,-23873,-34927,6963,85487,78047
C00725=-93466,-23543,-36325,6911,86486,78200
C00726=-93670,-22147,-39411,6941,89101,78276
C00727=-92980,-26767,-42567,6357,64758,77223
C00728=-92830,-24983,-37315,6405,62444,77148
C00729=-92885,-24260,-35203,6486,61526,77076
C00730=-95062,-23529,-34681,8624,61962,76228
C00731=-95090,-24132,-36711,8569,62895,76288
C00732=-95328,-25868,-41938,8524,65219,76375
C00733=-95261,-25907,-41974,7480,65026,76408
C00734=-95085,-24145,-36729,7536,62706,76321
C00735=-95201,-23568,-34719,7655,61783,76214
C00736=-93539,-24230,-35181,6102,61462,76860
C00737=-92783,-25001,-37319,5340,62272,77201
C00738=-92870,-26808,-42587,5281,64581,77276
C00739=-120452,-88146,-86102,21652,66713,67139
C00740=-165262,-16782,-33522,47685,80918,53825
C00741=-161018,-5245,-12472,47809,73866,52405
C00742=-160589,-4232,-10187,47903,73032,52200
C00743=-158091,-13363,-17379,47446,71525,52709
C00744=-158239,-15440,-20419,47297,72158,52954
C00745=-159752,-17175,-25374,47188,74446,53337
C00746=-148723,45367,2700,12479,106062,61188
C00747=-148955,42713,4001,12346,103979,60892
C00748=-149715,44338,7129,12324,103024,60537
C00749=-146495,33091,-4314,12210,103798,61708
C00750=-146015,32884,-6147,12245,104729,61965
C00751=-145791,35660,-7470,12388,106889,62265
C00752=-109011,-26713,-50438,8452,98222,74634
C00753=-84134,-123556,-96733,5664,74963,81774
C00754=-10907,-117335,-90652,-18762,63715,-59495
BC00000=165820,667836,1075229
BC00001=35816,1008911,1075175
BC00002=35816,1008911,1075175
BC00003=35816,1008911,1075175
BC00004=35816,1008911,1075175
BC00005=35816,1008911,1075175
BC00006=35816,1008911,1075175
BC00007=35816,1008911,1075175
BC00008=35816,1008911,1075175
BC00009=81778,1000994,1075175
BC00010=81778,1000994,1075175
BC00011=81778,1000994,1075175
BC00012=81778,1000994,1075175
BC00013=81778,1000994,1075175
BC00014=81778,1000994,1075175
BC00015=81778,1000994,1075175
BC00016=81778,1000994,1075175
BC00017=183238,908205,1075175
BC00018=183238,908205,1075175
BC00019=183238,908205,1075175
BC00020=183238,908205,1075175
BC00021=183238,908205,1075175
BC00022=183238,908205,1075175
BC00023=183238,908205,1075175
BC00024=183238,908205,1075175
BC00025=183238,908205,1075175
BC00026=183238,908205,1075175
BC00027=183238,908205,1075175
BC00028=183238,908205,1075175
BC00029=183238,908205,1075175
BC00030=183238,908205,1075175
BC00031=277080,941460,1075175
BC00032=289789,946711,1075175
BC00033=289789,946711,1075175
BC00034=289789,946711,1075175
BC00035=289789,946711,1075175
BC00036=289789,946711,1075175
BC00037=289789,946711,1075175
BC00038=289789,946711,1075175
BC00039=289789,946711,1075175
BC00040=289789,946711,1075175
BC00041=289789,946711,1075175
BC00042=289789,946711,1075175
BC00043=289789,946711,1075175
BC00044=289789,946711,1075175
BC00045=261300,945494,1075175
BC00046=261300,945494,1075175
BC00047=261300,945494,1075175
BC00048=261300,945494,1075175
BC00049=261300,945494,1075175
BC00050=261300,945494,1075175
BC00051=261300,945494,1075175
BC00052=261300,945494,1075175
BC00053=261300,945494,1075175
BC00054=261300,945494,1075175
BC00055=261300,945494,1075175
BC00056=261300,945494,1075175
BC00057=261300,945494,1075175
BC00058=293747,972847,1075175
BC00059=293747,972847,1075175
BC00060=293747,972847,1075175
BC00061=293747,972847,1075175
BC00062=293747,972847,1075175
BC00063=293747,972847,1075175
BC00064=293747,972847,1075175
BC00065=293747,972847,1075175
BC00066=293747,958005,1075175
BC00067=262329,883284,1075175
BC00068=265687,860722,1075175
BC00069=265687,860722,1075175
BC00070=265687,860722,1075175
BC00071=265687,860722,1075175
BC00072=265687,860722,1075175
BC00073=265687,860722,1075175
BC00074=265687,860722,1075175
BC00075=265687,860722,1075175
BC00076=265687,860722,1075175
BC00077=265687,860722,1075175
BC00078=265687,860722,1075175
BC00079=265687,860722,1075175
BC00080=265687,860722,1075175
BC00081=272052,840663,1075175
BC00082=272052,840663,1075175
BC00083=272052,840663,1075175
BC00084=272052,840663,1075175
BC00085=272052,840663,1075175
BC00086=272052,840663,1075175
BC00087=272052,840663,1075175
BC00088=272052,840663,1075175
BC00089=272052,840663,1075175
BC00090=294078,933568,1075175
BC00091=294078,933568,1075175
BC00092=294078,933568,1075175
BC00093=294078,933568,1075175
BC00094=294078,933568,1075175
BC00095=294078,933568,1075175
BC00096=294078,933568,1075175
BC00097=294078,933568,1075175
BC00098=294078,933568,1075175
BC00099=294078,933568,1075175
BC00100=294078,933568,1075175
BC00101=294078,933568,1075175
BC00102=294078,933568,1075175
BC00103=350010,851645,1075175
BC00104=398174,950083,1075175
BC00105=398174,950083,1075175
BC00106=398174,950083,1075175
BC00107=398174,950083,1075175
BC00108=398174,950083,1075175
BC00109=398174,950083,1075175
BC00110=398174,950083,1075175
BC00111=398174,950083,1075175
BC00112=398174,954074,1075175
BC00113=398174,954074,1075175
BC00114=398174,954074,1075175
BC00115=398174,954074,1075175
BC00116=398174,954074,1075175
BC00117=398174,954074,1075175
BC00118=398174,954074,1075175
BC00119=398174,954074,1075175
BC00120=398174,954074,1075175
BC00121=398174,870681,1075175
BC00122=398174,817728,1075175
BC00123=398174,817728,1075175
BC00124=398174,817728,1075175
BC00125=398174,817728,1075175
BC00126=398174,817728,1075175
BC00127=398174,817728,1075175
BC00128=398174,817728,1075175
BC00129=398174,817728,1075175
BC00130=398174,817728,1075175
BC00131=398174,817728,1075175
BC00132=398174,817728,1075175
BC00133=396448,827169,1075175
BC00134=394822,829620,1075175
BC00135=394822,829620,1075175
BC00136=394822,829620,1075175
BC00137=394822,829620,1075175
BC00138=394822,829620,1075175
BC00139=394822,829620,1075175
BC00140=394822,829620,1075175
BC00141=394822,829620,1075175
BC00142=394822,829620,1075175
BC00143=394822,829620,1075175
BC00144=394822,829620,1075175
BC00145=355383,833896,1075175
BC00146=324600,845042,1075175
BC00147=324600,845042,1075175
BC00148=324600,845042,1075175
BC00149=324600,845042,1075175
BC00150=324600,845042,1075175
BC00151=324600,845042,1075175
BC00152=324600,845042,1075175
BC00153=324600,845042,1075175
BC00154=311941,807883,1075175
BC00155=311941,807883,1075175
BC00156=311941,807883,1075175
BC00157=311941,807883,1075175
BC00158=311941,807883,1075175
BC00159=311941,807883,1075175
BC00160=311941,807883,1075175
BC00161=311941,807883,1075175
BC00162=311941,807883,1075175
BC00163=311941,807883,1075175
BC00164=311941,807883,1075175
BC00165=311941,807883,1075175
BC00166=316281,962914,1075175
BC00167=312573,990264,1075175
BC00168=307903,987774,1075175
BC00169=306034,986778,1075175
BC00170=306034,986778,1075175
BC00171=306034,986778,1075175
BC00172=283260,992694,1075175
BC00173=316930,973741,1075175
BC00174=283185,985095,1075172
BC00175=281644,987513,1075175
BC00176=279107,993102,1075175
BC00177=280151,960541,1075175
BC00178=281317,877250,1075175
BC00179=282638,819792,1075175
BC00180=284858,824834,1075175
BC00181=285747,826851,1075175
BC00182=285747,826851,1075175
BC00183=285747,826851,1075175
BC00184=239186,852971,1075175
BC00185=275413,838907,1075175
BC00186=285600,832969,1075175
BC00187=288466,826898,1075175
BC00188=288466,826898,1075175
BC00189=136054,1003977,1075175
BC00190=136349,1009357,1075175
BC00191=136467,1011509,1075175
BC00192=85590,1020321,1075175
BC00193=85472,1018169,1075175
BC00194=85177,1012789,1075175
BC00195=85177,867663,1075175
BC00196=394575,855601,1075175
BC00197=335365,938803,1075175
BC00198=336708,934958,1075175
BC00199=337245,935767,1075175
BC00200=337268,942708,1075175
BC00201=336730,941898,1075175
BC00202=295940,927161,1075175
BC00203=295940,927161,1075175
BC00204=295940,927161,1075175
BC00205=295940,927161,1075175
BC00206=295940,927161,1075175
BC00207=295940,927161,1075175
BC00208=295940,927161,1075175
BC00209=295940,927161,1075175
BC00210=393681,912027,1075175
BC00211=398174,921728,1075175
BC00212=398174,926962,1075175
BC00213=398174,928620,1075175
BC00214=364761,938622,1075175
BC00215=369199,937365,1075175
BC00216=369642,935240,1075175
BC00217=370750,929927,1075175
BC00218=370750,848394,1075175
BC00219=340693,834439,1075175
BC00220=313140,829466,1075175
BC00221=312428,824087,1075175
BC00222=312144,821935,1075175
BC00223=307365,821950,1075175
BC00224=268115,822068,1075172
BC00225=280175,821658,1075175
BC00226=281271,823684,1075175
BC00227=284011,828752,1075175
BC00228=290728,897938,1075175
BC00229=293762,929183,1075175
BC00230=290448,934424,1075175
BC00231=289122,936520,1075175
BC00232=241729,942952,1075175
BC00233=279832,936352,1075175
BC00234=264136,939681,1075175
BC00235=262547,937931,1075175
BC00236=258574,933557,1075175
BC00237=314949,872913,1075175
BC00238=378471,827894,1075175
BC00239=380915,822749,1075175
BC00240=381893,820691,1075175
BC00241=398174,825891,1075175
BC00242=361449,826034,1075175
BC00243=398174,815367,1075175
BC00244=398174,817132,1075175
BC00245=398174,821543,1075175
BC00246=398174,821543,1075175
BC00247=256492,965748,1075175
BC00248=237924,1001427,1075175
BC00249=237924,1015453,1075175
BC00250=232933,1013664,1075175
BC00251=230937,1012949,1075175
BC00252=178459,1050835,1075175
BC00253=213013,1031453,1075175
BC00254=227041,1020134,1075175
BC00255=235513,1004484,1075175
BC00256=237128,986927,1075175
BC00257=233266,973358,1075175
BC00258=228054,964181,1075175
BC00259=223178,957936,1075175
BC00260=220682,955545,1075175
BC00261=222343,954677,1075175
BC00262=225664,952941,1075175
BC00263=141848,914666,1075175
BC00264=143128,920299,1075175
BC00265=143639,922553,1075175
BC00266=137651,924704,1075175
BC00267=129694,927561,1075175
BC00268=134120,930846,1075175
BC00269=148671,926943,1075175
BC00270=116938,942468,1075175
BC00271=115693,943064,1075175
BC00272=111414,945116,1075175
BC00273=111414,945116,1075175
BC00274=111414,945116,1075175
BC00275=110923,942951,1075175
BC00276=109940,938621,1075175
BC00277=131749,675704,1075175
BC00278=165820,667836,1075229
BC00279=35816,1008911,1075175
BC00280=35816,1008911,1075175
BC00281=35816,1008911,1075175
BC00282=35816,1008911,1075175
BC00283=35816,1008911,1075175
BC00284=35816,1008911,1075175
BC00285=35816,1008911,1075175
BC00286=35816,1008911,1075175
BC00287=81778,1000994,1075175
BC00288=81778,1000994,1075175
BC00289=81778,1000994,1075175
BC00290=81778,1000994,1075175
BC00291=81778,1000994,1075175
BC00292=81778,1000994,1075175
BC00293=81778,1000994,1075175
BC00294=81778,1000994,1075175
BC00295=183238,908205,1075175
BC00296=183238,908205,1075175
BC00297=183238,908205,1075175
BC00298=183238,908205,1075175
BC00299=183238,908205,1075175
BC00300=183238,908205,1075175
BC00301=183238,908205,1075175
BC00302=183238,908205,1075175
BC00303=183238,908205,1075175
BC00304=183238,908205,1075175
BC00305=183238,908205,1075175
BC00306=183238,908205,1075175
BC00307=183238,908205,1075175
BC00308=183238,908205,1075175
BC00309=277080,941460,1075175
BC00310=289789,946711,1075175
BC00311=289789,946711,1075175
BC00312=289789,946711,1075175
BC00313=289789,946711,1075175
BC00314=289789,946711,1075175
BC00315=289789,946711,1075175
BC00316=289789,946711,1075175
BC00317=289789,946711,1075175
BC00318=289789,946711,1075175
BC00319=289789,946711,1075175
BC00320=289789,946711,1075175
BC00321=289789,946711,1075175
BC00322=289789,946711,1075175
BC00323=261300,945494,1075175
BC00324=261300,945494,1075175
BC00325=261300,945494,1075175
BC00326=261300,945494,1075175
BC00327=261300,945494,1075175
BC00328=261300,945494,1075175
BC00329=261300,945494,1075175
BC00330=261300,945494,1075175
BC00331=261300,945494,1075175
BC00332=261300,945494,1075175
BC00333=261300,945494,1075175
BC00334=261300,945494,1075175
BC00335=261300,945494,1075175
BC00336=293747,972847,1075175
BC00337=293747,972847,1075175
BC00338=293747,972847,1075175
BC00339=293747,972847,1075175
BC00340=293747,972847,1075175
BC00341=293747,972847,1075175
BC00342=293747,972847,1075175
BC00343=293747,972847,1075175
BC00344=293747,958005,1075175
BC00345=262329,883284,1075175
BC00346=265687,860722,1075175
BC00347=265687,860722,1075175
BC00348=265687,860722,1075175
BC00349=265687,860722,1075175
BC00350=265687,860722,1075175
BC00351=265687,860722,1075175
BC00352=265687,860722,1075175
BC00353=265687,860722,1075175
BC00354=265687,860722,1075175
BC00355=265687,860722,1075175
BC00356=265687,860722,1075175
BC00357=265687,860722,1075175
BC00358=265687,860722,1075175
BC00359=272052,840663,1075175
BC00360=272052,840663,1075175
BC00361=272052,840663,1075175
BC00362=272052,840663,1075175
BC00363=272052,840663,1075175
BC00364=272052,840663,1075175
BC00365=272052,840663,1075175
BC00366=272052,840663,1075175
BC00367=272052,840663,1075175
BC00368=294078,933568,1075175
BC00369=294078,933568,1075175
BC00370=294078,933568,1075175
BC00371=294078,933568,1075175
BC00372=294078,933568,1075175
BC00373=294078,933568,1075175
BC00374=294078,933568,1075175
BC00375=294078,933568,1075175
BC00376=294078,933568,1075175
BC00377=294078,933568,1075175
BC00378=294078,933568,1075175
BC00379=294078,933568,1075175
BC00380=294078,933568,1075175
BC00381=350010,851645,1075175
BC00382=398174,950083,1075175
BC00383=398174,950083,1075175
BC00384=398174,950083,1075175
BC00385=398174,950083,1075175
BC00386=398174,950083,1075175
BC00387=398174,950083,1075175
BC00388=398174,950083,1075175
BC00389=398174,950083,1075175
BC00390=398174,954074,1075175
BC00391=398174,954074,1075175
BC00392=398174,954074,1075175
BC00393=398174,954074,1075175
BC00394=398174,954074,1075175
BC00395=398174,954074,1075175
BC00396=398174,954074,1075175
BC00397=398174,954074,1075175
BC00398=398174,954074,1075175
BC00399=398174,870681,1075175
BC00400=398174,817728,1075175
BC00401=398174,817728,1075175
BC00402=398174,817728,1075175
BC00403=398174,817728,1075175
BC00404=398174,817728,1075175
BC00405=398174,817728,1075175
BC00406=398174,817728,1075175
BC00407=398174,817728,1075175
BC00408=398174,817728,1075175
BC00409=398174,817728,1075175
BC00410=398174,817728,1075175
BC00411=396448,827169,1075175
BC00412=394822,829620,1075175
BC00413=394822,829620,1075175
BC00414=394822,829620,1075175
BC00415=394822,829620,1075175
BC00416=394822,829620,1075175
BC00417=394822,829620,1075175
BC00418=394822,829620,1075175
BC00419=394822,829620,1075175
BC00420=394822,829620,1075175
BC00421=394822,829620,1075175
BC00422=394822,829620,1075175
BC00423=355383,833896,1075175
BC00424=324600,845042,1075175
BC00425=324600,845042,1075175
BC00426=324600,845042,1075175
BC00427=324600,845042,1075175
BC00428=324600,845042,1075175
BC00429=324600,845042,1075175
BC00430=324600,845042,1075175
BC00431=324600,845042,1075175
BC00432=311941,807883,1075175
BC00433=311941,807883,1075175
BC00434=311941,807883,1075175
BC00435=311941,807883,1075175
BC00436=311941,807883,1075175
BC00437=311941,807883,1075175
BC00438=311941,807883,1075175
BC00439=311941,807883,1075175
BC00440=311941,807883,1075175
BC00441=311941,807883,1075175
BC00442=311941,807883,1075175
BC00443=311941,807883,1075175
BC00444=316281,962914,1075175
BC00445=312573,990264,1075175
BC00446=307903,987774,1075175
BC00447=306034,986778,1075175
BC00448=306034,986778,1075175
BC00449=306034,986778,1075175
BC00450=283260,992694,1075175
BC00451=316930,973741,1075175
BC00452=283185,985095,1075172
BC00453=281644,987513,1075175
BC00454=279107,993102,1075175
BC00455=280151,960541,1075175
BC00456=281317,877250,1075175
BC00457=282638,819792,1075175
BC00458=284858,824834,1075175
BC00459=285747,826851,1075175
BC00460=285747,826851,1075175
BC00461=285747,826851,1075175
BC00462=239186,852971,1075175
BC00463=275413,838907,1075175
BC00464=285600,832969,1075175
BC00465=288466,826898,1075175
BC00466=288466,826898,1075175
BC00467=136054,1003977,1075175
BC00468=136349,1009357,1075175
BC00469=136467,1011509,1075175
BC00470=85590,1020321,1075175
BC00471=85472,1018169,1075175
BC00472=85177,1012789,1075175
BC00473=85177,867663,1075175
BC00474=394575,855601,1075175
BC00475=335365,938803,1075175
BC00476=336708,934958,1075175
BC00477=337245,935767,1075175
BC00478=337268,942708,1075175
BC00479=336730,941898,1075175
BC00480=295940,927161,1075175
BC00481=295940,927161,1075175
BC00482=295940,927161,1075175
BC00483=295940,927161,1075175
BC00484=295940,927161,1075175
BC00485=295940,927161,1075175
BC00486=295940,927161,1075175
BC00487=295940,927161,1075175
BC00488=393681,912027,1075175
BC00489=398174,921728,1075175
BC00490=398174,926962,1075175
BC00491=398174,928620,1075175
BC00492=364761,938622,1075175
BC00493=369199,937365,1075175
BC00494=369642,935240,1075175
BC00495=370750,929927,1075175
BC00496=370750,848394,1075175
BC00497=340693,834439,1075175
BC00498=313140,829466,1075175
BC00499=312428,824087,1075175
BC00500=312144,821935,1075175
BC00501=307365,821950,1075175
BC00502=268115,822068,1075172
BC00503=280175,821657,1075175
BC00504=281271,823684,1075175
BC00505=284011,828752,1075175
BC00506=290728,897938,1075175
BC00507=293762,929183,1075175
BC00508=290448,934424,1075175
BC00509=289122,936520,1075175
BC00510=241729,942952,1075175
BC00511=279832,936352,1075175
BC00512=264136,939681,1075175
BC00513=262547,937931,1075175
BC00514=258574,933557,1075175
BC00515=314949,872913,1075175
BC00516=378471,827894,1075175
BC00517=380915,822749,1075175
BC00518=381893,820691,1075175
BC00519=398174,825891,1075175
BC00520=361449,826034,1075175
BC00521=398174,815367,1075175
BC00522=398174,817132,1075175
BC00523=398174,821543,1075175
BC00524=398174,821543,1075175
BC00525=256492,965748,1075175
BC00526=237924,1001427,1075175
BC00527=237924,1015453,1075175
BC00528=232933,1013664,1075175
BC00529=230937,1012949,1075175
BC00530=178459,1050835,1075175
BC00531=213013,1031453,1075175
BC00532=227041,1020134,1075175
BC00533=235513,1004484,1075175
BC00534=237128,986927,1075175
BC00535=233266,973358,1075175
BC00536=228054,964181,1075175
BC00537=223178,957936,1075175
BC00538=220682,955545,1075175
BC00539=222343,954677,1075175
BC00540=225664,952941,1075175
BC00541=141848,914666,1075175
BC00542=143128,920299,1075175
BC00543=148671,926943,1075175
BC00544=143639,922553,1075175
BC00545=137651,924704,1075175
BC00546=129694,927561,1075175
BC00547=134120,930846,1075175
BC00548=148671,926943,1075175
BC00549=116938,942468,1075175
BC00550=115693,943064,1075175
BC00551=111414,945116,1075175
BC00552=111414,945116,1075175
BC00553=111414,945116,1075175
BC00554=110923,942951,1075175
BC00555=109940,938621,1075175
BC00556=131749,675704,1075175
BC00557=21214,672831,429902
BC00558=66815,724118,419761
BC00559=110240,772957,337669
BC00560=136729,789553,283981
BC00561=136729,789553,283981
BC00562=136729,789553,283981
BC00563=136729,789553,283981
BC00564=136729,789553,283981
BC00565=136729,789553,283981
BC00566=136729,789553,283981
BC00567=136729,789553,283981
BC00568=136729,789553,283981
BC00569=163194,789553,386705
BC00570=163194,789553,386705
BC00571=163194,789553,386705
BC00572=163194,789553,386705
BC00573=163194,789553,386705
BC00574=163194,789553,386705
BC00575=163194,789553,386705
BC00576=163194,789553,386705
BC00577=163194,789553,386705
BC00578=110240,772957,337669
BC00579=66815,724118,419761
BC00580=66815,670858,419761
BC00581=252765,670858,277331
BC00582=322808,760288,131711
BC00583=322808,760288,131711
BC00584=322808,760288,131711
BC00585=322808,760288,131711
BC00586=322808,760288,131711
BC00587=322808,760288,131711
BC00588=322808,760288,131711
BC00589=322808,760288,131711
BC00590=322808,760288,131711
BC00591=340407,752653,125690
BC00592=340407,752653,125690
BC00593=340407,752653,125690
BC00594=340407,752653,125690
BC00595=340407,752653,125690
BC00596=340407,752653,125690
BC00597=340407,752653,125690
BC00598=340407,752653,125690
BC00599=309477,783812,200910
BC00600=309477,783812,200910
BC00601=309477,783812,200910
BC00602=309477,783812,200910
BC00603=309477,783812,200910
BC00604=309477,783812,200910
BC00605=309477,783812,200910
BC00606=309477,783812,200910
BC00607=309477,783812,200910
BC00608=309477,783812,200910
BC00609=309477,783812,200910
BC00610=309477,783812,200910
BC00611=335534,789553,204922
BC00612=335534,789553,204922
BC00613=335534,789553,204922
BC00614=335534,789553,204922
BC00615=335534,789553,204922
BC00616=335534,789553,204922
BC00617=335534,789553,204922
BC00618=335534,789553,204922
BC00619=335534,789553,204922
BC00620=344006,752651,139062
BC00621=344006,752651,139062
BC00622=344006,752651,139062
BC00623=344006,752651,139062
BC00624=344006,752651,139062
BC00625=344006,752651,139062
BC00626=344006,752651,139062
BC00627=344006,752651,139062
BC00628=344006,752651,139062
BC00629=374489,733638,136084
BC00630=374489,733638,136084
BC00631=374489,733638,136084
BC00632=374489,733638,136084
BC00633=374489,733638,136084
BC00634=374489,733638,136084
BC00635=374489,733638,136084
BC00636=374489,733638,136084
BC00637=374489,733638,136084
BC00638=300933,750795,218908
BC00639=283893,750061,250495
BC00640=276320,749735,264534
BC00641=276320,749735,264534
BC00642=276320,749735,264534
BC00643=276320,749735,264534
BC00644=276320,749735,264534
BC00645=276320,749735,264534
BC00646=276320,749735,264534
BC00647=276320,749735,264534
BC00648=276320,749735,264534
BC00649=248857,763770,138691
BC00650=248857,763770,138691
BC00651=248857,763770,138691
BC00652=248857,763770,138691
BC00653=248857,763770,138691
BC00654=248857,763770,138691
BC00655=248857,763770,138691
BC00656=248857,763770,138691
BC00657=248857,763770,138691
BC00658=248857,763770,138691
BC00659=315051,758770,94341
BC00660=315051,758770,94341
BC00661=315051,758770,94341
BC00662=315051,758770,94341
BC00663=315051,758770,94341
BC00664=315051,758770,94341
BC00665=315051,758770,94341
BC00666=315051,758770,94341
BC00667=315051,758770,94341
BC00668=315051,758770,94341
BC00669=398174,761952,129173
BC00670=398174,761952,129173
BC00671=398174,761952,129173
BC00672=398174,761952,129173
BC00673=398174,761952,129173
BC00674=398174,761952,129173
BC00675=366295,778309,120132
BC00676=366295,778309,120132
BC00677=366295,778309,120132
BC00678=366295,778309,120132
BC00679=366295,778309,120132
BC00680=366295,778309,120132
BC00681=398174,729290,94227
BC00682=398174,729290,94227
BC00683=398174,729290,94227
BC00684=398174,729290,94227
BC00685=398174,729290,94227
BC00686=398174,729290,94227
BC00687=382568,752165,121199
BC00688=382568,752165,121199
BC00689=382568,752165,121199
BC00690=382568,752165,121199
BC00691=382568,752165,121199
BC00692=382568,752165,121199
BC00693=382568,668969,422236
BC00694=167343,668969,639457
BC00695=112241,789553,268043
BC00696=112241,789553,268043
BC00697=112241,789553,268043
BC00698=112241,789553,268043
BC00699=112241,789553,268043
BC00700=112241,789553,268043
BC00701=121114,789553,252467
BC00702=121114,789553,252467
BC00703=121114,789553,252467
BC00704=121114,789553,252467
BC00705=121114,789553,252467
BC00706=121114,789553,252467
BC00707=121337,789553,329708
BC00708=121337,789553,329708
BC00709=121337,789553,329708
BC00710=121337,789553,329708
BC00711=121337,789553,329708
BC00712=121337,789553,329708
BC00713=167343,668969,639457
BC00714=382568,668969,422236
BC00715=299251,773200,237241
BC00716=299251,773200,237241
BC00717=299251,773200,237241
BC00718=299251,773200,237241
BC00719=299251,773200,237241
BC00720=299251,773200,237241
BC00721=279478,784302,237667
BC00722=279478,784302,237667
BC00723=279478,784302,237667
BC00724=279478,784302,237667
BC00725=279478,784302,237667
BC00726=279478,784302,237667
BC00727=280278,760811,181687
BC00728=280278,760811,181687
BC00729=280278,760811,181687
BC00730=280278,760811,181687
BC00731=280278,760811,181687
BC00732=280278,760811,181687
BC00733=277549,762343,181693
BC00734=277549,762343,181693
BC00735=277549,762343,181693
BC00736=277549,762343,181693
BC00737=277549,762343,181693
BC00738=277549,762343,181693
BC00739=297275,771567,184324
BC00740=335741,789553,189453
BC00741=335741,789553,189453
BC00742=335741,789553,189453
BC00743=335741,789553,189453
BC00744=335741,789553,189453
BC00745=335741,789553,189453
BC00746=351391,768330,121496
BC00747=351391,768330,121496
BC00748=351391,768330,121496
BC00749=351391,768330,121496
BC00750=351391,768330,121496
BC00751=351391,768330,121496
BC00752=283893,750061,250495
BC00753=283893,750061,250495
BC00754=165820,667836,534036
EC00000=798156,1112951
EC00001=798156,1112951
EC00002=798156,1112951
EC00003=798156,1112951
EC00004=798156,1112951
EC00005=798156,1112951
EC00006=798156,1112951
EC00007=798156,1112951
EC00008=798156,1112951
EC00009=798156,1112951
EC00010=798156,1112951
EC00011=798156,1112951
EC00012=798156,1112951
EC00013=798156,1112951
EC00014=798156,1112951
EC00015=798156,1112951
EC00016=798156,1112951
EC00017=798156,1112951
EC00018=798156,1112951
EC00019=798156,1112951
EC00020=798156,1112951
EC00021=798156,1112951
EC00022=798156,1112951
EC00023=798156,1112951
EC00024=798156,1112951
EC00025=798156,1112951
EC00026=798156,1112951
EC00027=798156,1112951
EC00028=798156,1112951
EC00029=798156,1112951
EC00030=798156,1112951
EC00031=798156,1112951
EC00032=798156,1112951
EC00033=798156,1112951
EC00034=798156,1112951
EC00035=798156,1112951
EC00036=798156,1112951
EC00037=798156,1112951
EC00038=798156,1112951
EC00039=798156,1112951
EC00040=798156,1112951
EC00041=798156,1112951
EC00042=798156,1112951
EC00043=798156,1112951
EC00044=798156,1112951
EC00045=798156,1112951
EC00046=798156,1112951
EC00047=798156,1112951
EC00048=798156,1112951
EC00049=798156,1112951
EC00050=798156,1112951
EC00051=798156,1112951
EC00052=798156,1112951
EC00053=798156,1112951
EC00054=798156,1112951
EC00055=798156,1112951
EC00056=798156,1112951
EC00057=798156,1112951
EC00058=798156,1112951
EC00059=798156,1112951
EC00060=798156,1112951
EC00061=798156,1112951
EC00062=798156,1112951
EC00063=798156,1112951
EC00064=798156,1112951
EC00065=798156,1112951
EC00066=798156,1112951
EC00067=798156,1112951
EC00068=798156,1112951
EC00069=798156,1112951
EC00070=798156,1112951
EC00071=798156,1112951
EC00072=798156,1112951
EC00073=798156,1112951
EC00074=798156,1112951
EC00075=798156,1112951
EC00076=798156,1112951
EC00077=798156,1112951
EC00078=798156,1112951
EC00079=798156,1112951
EC00080=798156,1112951
EC00081=798156,1112951
EC00082=798156,1112951
EC00083=798156,1112951
EC00084=798156,1112951
EC00085=798156,1112951
EC00086=798156,1112951
EC00087=798156,1112951
EC00088=798156,1112951
EC00089=798156,1112951
EC00090=798156,1112951
EC00091=798156,1112951
EC00092=798156,1112951
EC00093=798156,1112951
EC00094=798156,1112951
EC00095=798156,1112951
EC00096=798156,1112951
EC00097=798156,1112951
EC00098=798156,1112951
EC00099=798156,1112951
EC00100=798156,1112951
EC00101=798156,1112951
EC00102=798156,1112951
EC00103=798156,1112951
EC00104=798156,1112951
EC00105=798156,1112951
EC00106=798156,1112951
EC00107=798156,1112951
EC00108=798156,1112951
EC00109=798156,1112951
EC00110=798156,1112951
EC00111=798156,1112951
EC00112=798156,1112951
EC00113=798156,1112951
EC00114=798156,1112951
EC00115=798156,1112951
EC00116=798156,1112951
EC00117=798156,1112951
EC00118=798156,1112951
EC00119=798156,1112951
EC00120=798156,1112951
EC00121=798156,1112951
EC00122=798156,1112951
EC00123=798156,1112951
EC00124=798156,1112951
EC00125=798156,1112951
EC00126=798156,1112951
EC00127=798156,1112951
EC00128=798156,1112951
EC00129=798156,1112951
EC00130=798156,1112951
EC00131=798156,1112951
EC00132=798156,1112951
EC00133=798156,1112951
EC00134=798156,1112951
EC00135=798156,1112951
EC00136=798156,1112951
EC00137=798156,1112951
EC00138=798156,1112951
EC00139=798156,1112951
EC00140=798156,1112951
EC00141=798156,1112951
EC00142=798156,1112951
EC00143=798156,1112951
EC00144=798156,1112951
EC00145=798156,1112951
EC00146=798156,1112951
EC00147=798156,1112951
EC00148=798156,1112951
EC00149=798156,1112951
EC00150=798156,1112951
EC00151=798156,1112951
EC00152=798156,1112951
EC00153=798156,1112951
EC00154=798156,1112951
EC00155=798156,1112951
EC00156=798156,1112951
EC00157=798156,1112951
EC00158=798156,1112951
EC00159=798156,1112951
EC00160=798156,1112951
EC00161=798156,1112951
EC00162=798156,1112951
EC00163=798156,1112951
EC00164=798156,1112951
EC00165=798156,1112951
EC00166=798156,1112951
EC00167=798156,1112951
EC00168=798156,1112951
EC00169=798156,1112951
EC00170=798156,1112951
EC00171=798156,1112951
EC00172=798156,1112951
EC00173=798156,1112951
EC00174=798155,1112950
EC00175=798156,1112951
EC00176=798156,1112951
EC00177=798156,1112951
EC00178=798156,1112951
EC00179=798156,1112951
EC00180=798156,1112951
EC00181=798156,1112951
EC00182=798156,1112951
EC00183=798156,1112951
EC00184=798156,1112951
EC00185=798156,1112951
EC00186=798156,1112951
EC00187=798156,1112951
EC00188=798156,1112951
EC00189=798156,1112951
EC00190=798156,1112951
EC00191=798156,1112951
EC00192=798156,1112951
EC00193=798156,1112951
EC00194=798156,1112951
EC00195=798156,1112951
EC00196=798156,1112951
EC00197=798156,1112951
EC00198=798156,1112951
EC00199=798156,1112951
EC00200=798156,1112951
EC00201=798156,1112951
EC00202=798156,1112951
EC00203=798156,1112951
EC00204=798156,1112951
EC00205=798156,1112951
EC00206=798156,1112951
EC00207=798156,1112951
EC00208=798156,1112951
EC00209=798156,1112951
EC00210=798156,1112951
EC00211=798156,1112951
EC00212=798156,1112951
EC00213=798156,1112951
EC00214=798156,1112951
EC00215=798156,1112951
EC00216=798156,1112951
EC00217=798156,1112951
EC00218=798156,1112951
EC00219=798156,1112951
EC00220=798156,1112951
EC00221=798156,1112951
EC00222=798156,1112951
EC00223=798156,1112951
EC00224=798155,1112950
EC00225=798156,1112950
EC00226=798156,1112951
EC00227=798156,1112951
EC00228=798156,1112951
EC00229=798156,1112951
EC00230=798156,1112951
EC00231=798156,1112951
EC00232=798156,1112951
EC00233=798156,1112951
EC00234=798156,1112951
EC00235=798156,1112951
EC00236=798156,1112951
EC00237=798156,1112951
EC00238=798156,1112951
EC00239=798156,1112951
EC00240=798156,1112951
EC00241=798156,1112951
EC00242=798156,1112951
EC00243=798156,1112951
EC00244=798156,1112951
EC00245=798156,1112951
EC00246=798156,1112951
EC00247=798156,1112951
EC00248=798156,1112951
EC00249=798156,1112951
EC00250=798156,1112951
EC00251=798156,1112951
EC00252=798156,1112951
EC00253=798156,1112951
EC00254=798156,1112951
EC00255=798156,1112951
EC00256=798156,1112951
EC00257=798156,1112951
EC00258=798156,1112951
EC00259=798156,1112951
EC00260=798156,1112951
EC00261=798156,1112951
EC00262=798156,1112951
EC00263=798156,1112951
EC00264=798156,1112951
EC00265=798156,1112951
EC00266=798156,1112951
EC00267=798156,1112951
EC00268=798156,1112951
EC00269=798156,1112951
EC00270=798156,1112951
EC00271=798156,1112951
EC00272=798156,1112951
EC00273=798156,1112951
EC00274=798156,1112951
EC00275=798156,1112951
EC00276=798156,1112951
EC00277=798156,1112951
EC00278=798156,1112951
EC00279=798156,1112951
EC00280=798156,1112951
EC00281=798156,1112951
EC00282=798156,1112951
EC00283=798156,1112951
EC00284=798156,1112951
EC00285=798156,1112951
EC00286=798156,1112951
EC00287=798156,1112951
EC00288=798156,1112951
EC00289=798156,1112951
EC00290=798156,1112951
EC00291=798156,1112951
EC00292=798156,1112951
EC00293=798156,1112951
EC00294=798156,1112951
EC00295=798156,1112951
EC00296=798156,1112951
EC00297=798156,1112951
EC00298=798156,1112951
EC00299=798156,1112951
EC00300=798156,1112951
EC00301=798156,1112951
EC00302=798156,1112951
EC00303=798156,1112951
EC00304=798156,1112951
EC00305=798156,1112951
EC00306=798156,1112951
EC00307=798156,1112951
EC00308=798156,1112951
EC00309=798156,1112951
EC00310=798156,1112951
EC00311=798156,1112951
EC00312=798156,1112951
EC00313=798156,1112951
EC00314=798156,1112951
EC00315=798156,1112951
EC00316=798156,1112951
EC00317=798156,1112951
EC00318=798156,1112951
EC00319=798156,1112951
EC00320=798156,1112951
EC00321=798156,1112951
EC00322=798156,1112951
EC00323=798156,1112951
EC00324=798156,1112951
EC00325=798156,1112951
EC00326=798156,1112951
EC00327=798156,1112951
EC00328=798156,1112951
EC00329=798156,1112951
EC00330=798156,1112951
EC00331=798156,1112951
EC00332=798156,1112951
EC00333=798156,1112951
EC00334=798156,1112951
EC00335=798156,1112951
EC00336=798156,1112951
EC00337=798156,1112951
EC00338=798156,1112951
EC00339=798156,1112951
EC00340=798156,1112951
EC00341=798156,1112951
EC00342=798156,1112951
EC00343=798156,1112951
EC00344=798156,1112951
EC00345=798156,1112951
EC00346=798156,1112951
EC00347=798156,1112951
EC00348=798156,1112951
EC00349=798156,1112951
EC00350=798156,1112951
EC00351=798156,1112951
EC00352=798156,1112951
EC00353=798156,1112951
EC00354=798156,1112951
EC00355=798156,1112951
EC00356=798156,1112951
EC00357=798156,1112951
EC00358=798156,1112951
EC00359=798156,1112951
EC00360=798156,1112951
EC00361=798156,1112951
EC00362=798156,1112951
EC00363=798156,1112951
EC00364=798156,1112951
EC00365=798156,1112951
EC00366=798156,1112951
EC00367=798156,1112951
EC00368=798156,1112951
EC00369=798156,1112951
EC00370=798156,1112951
EC00371=798156,1112951
EC00372=798156,1112951
EC00373=798156,1112951
EC00374=798156,1112951
EC00375=798156,1112951
EC00376=798156,1112951
EC00377=798156,1112951
EC00378=798156,1112951
EC00379=798156,1112951
EC00380=798156,1112951
EC00381=798156,1112951
EC00382=798156,1112951
EC00383=798156,1112951
EC00384=798156,1112951
EC00385=798156,1112951
EC00386=798156,1112951
EC00387=798156,1112951
EC00388=798156,1112951
EC00389=798156,1112951
EC00390=798156,1112951
EC00391=798156,1112951
EC00392=798156,1112951
EC00393=798156,1112951
EC00394=798156,1112951
EC00395=798156,1112951
EC00396=798156,1112951
EC00397=798156,1112951
EC00398=798156,1112951
EC00399=798156,1112951
EC00400=798156,1112951
EC00401=798156,1112951
EC00402=798156,1112951
EC00403=798156,1112951
EC00404=798156,1112951
EC00405=798156,1112951
EC00406=798156,1112951
EC00407=798156,1112951
EC00408=798156,1112951
EC00409=798156,1112951
EC00410=798156,1112951
EC00411=798156,1112951
EC00412=798156,1112951
EC00413=798156,1112951
EC00414=798156,1112951
EC00415=798156,1112951
EC00416=798156,1112951
EC00417=798156,1112951
EC00418=798156,1112951
EC00419=798156,1112951
EC00420=798156,1112951
EC00421=798156,1112951
EC00422=798156,1112951
EC00423=798156,1112951
EC00424=798156,1112951
EC00425=798156,1112951
EC00426=798156,1112951
EC00427=798156,1112951
EC00428=798156,1112951
EC00429=798156,1112951
EC00430=798156,1112951
EC00431=798156,1112951
EC00432=798156,1112951
EC00433=798156,1112951
EC00434=798156,1112951
EC00435=798156,1112951
EC00436=798156,1112951
EC00437=798156,1112951
EC00438=798156,1112951
EC00439=798156,1112951
EC00440=798156,1112951
EC00441=798156,1112951
EC00442=798156,1112951
EC00443=798156,1112951
EC00444=798156,1112951
EC00445=798156,1112951
EC00446=798156,1112951
EC00447=798156,1112951
EC00448=798156,1112951
EC00449=798156,1112951
EC00450=798156,1112951
EC00451=798156,1112951
EC00452=798155,1112950
EC00453=798156,1112951
EC00454=798156,1112951
EC00455=798156,1112951
EC00456=798156,1112951
EC00457=798156,1112951
EC00458=798156,1112951
EC00459=798156,1112951
EC00460=798156,1112951
EC00461=798156,1112951
EC00462=798156,1112951
EC00463=798156,1112951
EC00464=798156,1112951
EC00465=798156,1112951
EC00466=798156,1112951
EC00467=798156,1112951
EC00468=798156,1112951
EC00469=798156,1112951
EC00470=798156,1112951
EC00471=798156,1112951
EC00472=798156,1112951
EC00473=798156,1112951
EC00474=798156,1112951
EC00475=798156,1112951
EC00476=798156,1112951
EC00477=798156,1112951
EC00478=798156,1112951
EC00479=798156,1112951
EC00480=798156,1112951
EC00481=798156,1112951
EC00482=798156,1112951
EC00483=798156,1112951
EC00484=798156,1112951
EC00485=798156,1112951
EC00486=798156,1112951
EC00487=798156,1112951
EC00488=798156,1112951
EC00489=798156,1112951
EC00490=798156,1112951
EC00491=798156,1112951
EC00492=798156,1112951
EC00493=798156,1112951
EC00494=798156,1112951
EC00495=798156,1112951
EC00496=798156,1112951
EC00497=798156,1112951
EC00498=798156,1112951
EC00499=798156,1112951
EC00500=798156,1112951
EC00501=798156,1112951
EC00502=798155,1112950
EC00503=798156,1112951
EC00504=798156,1112951
EC00505=798156,1112951
EC00506=798156,1112951
EC00507=798156,1112951
EC00508=798156,1112951
EC00509=798156,1112951
EC00510=798156,1112951
EC00511=798156,1112951
EC00512=798156,1112951
EC00513=798156,1112951
EC00514=798156,1112951
EC00515=798156,1112951
EC00516=798156,1112951
EC00517=798156,1112951
EC00518=798156,1112951
EC00519=798156,1112951
EC00520=798156,1112951
EC00521=798156,1112951
EC00522=798156,1112951
EC00523=798156,1112951
EC00524=798156,1112951
EC00525=798156,1112951
EC00526=798156,1112951
EC00527=798156,1112951
EC00528=798156,1112951
EC00529=798156,1112951
EC00530=798156,1112951
EC00531=798156,1112951
EC00532=798156,1112951
EC00533=798156,1112951
EC00534=798156,1112951
EC00535=798156,1112951
EC00536=798156,1112951
EC00537=798156,1112951
EC00538=798156,1112951
EC00539=798156,1112951
EC00540=798156,1112951
EC00541=798156,1112951
EC00542=798156,1112951
EC00543=798156,1112951
EC00544=798156,1112951
EC00545=798156,1112951
EC00546=798156,1112951
EC00547=798156,1112951
EC00548=798156,1112951
EC00549=798156,1112951
EC00550=798156,1112951
EC00551=798156,1112951
EC00552=798156,1112951
EC00553=798156,1112951
EC00554=798156,1112951
EC00555=798156,1112951
EC00556=798156,1112951
EC00557=798156,1112951
EC00558=798156,1112951
EC00559=798156,1112951
EC00560=798156,1112951
EC00561=798156,1112951
EC00562=798156,1112951
EC00563=798156,1112951
EC00564=798156,1112951
EC00565=798156,1112951
EC00566=798156,1112951
EC00567=798156,1112951
EC00568=798156,1112951
EC00569=798156,1112951
EC00570=798156,1112951
EC00571=798156,1112951
EC00572=798156,1112951
EC00573=798156,1112951
EC00574=798156,1112951
EC00575=798156,1112951
EC00576=798156,1112951
EC00577=798156,1112951
EC00578=798156,1112951
EC00579=798156,1112951
EC00580=798156,1112951
EC00581=798156,1112951
EC00582=798156,1112951
EC00583=798156,1112951
EC00584=798156,1112951
EC00585=798156,1112951
EC00586=798156,1112951
EC00587=798156,1112951
EC00588=798156,1112951
EC00589=798156,1112951
EC00590=798156,1112951
EC00591=798156,1112951
EC00592=798156,1112951
EC00593=798156,1112951
EC00594=798156,1112951
EC00595=798156,1112951
EC00596=798156,1112951
EC00597=798156,1112951
EC00598=798156,1112951
EC00599=798156,1112951
EC00600=798156,1112951
EC00601=798156,1112951
EC00602=798156,1112951
EC00603=798156,1112951
EC00604=798156,1112951
EC00605=798156,1112951
EC00606=798156,1112951
EC00607=798156,1112951
EC00608=798156,1112951
EC00609=798156,1112951
EC00610=798156,1112951
EC00611=798156,1112951
EC00612=798156,1112951
EC00613=798156,1112951
EC00614=798156,1112951
EC00615=798156,1112951
EC00616=798156,1112951
EC00617=798156,1112951
EC00618=798156,1112951
EC00619=798156,1112951
EC00620=798156,1112951
EC00621=798156,1112951
EC00622=798156,1112951
EC00623=798156,1112951
EC00624=798156,1112951
EC00625=798156,1112951
EC00626=798156,1112951
EC00627=798156,1112951
EC00628=798156,1112951
EC00629=798156,1112951
EC00630=798156,1112951
EC00631=798156,1112951
EC00632=798156,1112951
EC00633=798156,1112951
EC00634=798156,1112951
EC00635=798156,1112951
EC00636=798156,1112951
EC00637=798156,1112951
EC00638=798156,1112951
EC00639=798156,1112951
EC00640=798156,1112951
EC00641=798156,1112951
EC00642=798156,1112951
EC00643=798156,1112951
EC00644=798156,1112951
EC00645=798156,1112951
EC00646=798156,1112951
EC00647=798156,1112951
EC00648=798156,1112951
EC00649=798156,1112951
EC00650=798156,1112951
EC00651=798156,1112951
EC00652=798156,1112951
EC00653=798156,1112951
EC00654=798156,1112951
EC00655=798156,1112951
EC00656=798156,1112951
EC00657=798156,1112951
EC00658=798156,1112951
EC00659=798156,1112951
EC00660=798156,1112951
EC00661=798156,1112951
EC00662=798156,1112951
EC00663=798156,1112951
EC00664=798156,1112951
EC00665=798156,1112951
EC00666=798156,1112951
EC00667=798156,1112951
EC00668=798156,1112951
EC00669=798156,1112951
EC00670=798156,1112951
EC00671=798156,1112951
EC00672=798156,1112951
EC00673=798156,1112951
EC00674=798156,1112951
EC00675=798156,1112951
EC00676=798156,1112951
EC00677=798156,1112951
EC00678=798156,1112951
EC00679=798156,1112951
EC00680=798156,1112951
EC00681=798156,1112951
EC00682=798156,1112951
EC00683=798156,1112951
EC00684=798156,1112951
EC00685=798156,1112951
EC00686=798156,1112951
EC00687=798156,1112951
EC00688=798156,1112951
EC00689=798156,1112951
EC00690=798156,1112951
EC00691=798156,1112951
EC00692=798156,1112951
EC00693=798156,1112951
EC00694=798156,1112951
EC00695=798156,1112951
EC00696=798156,1112951
EC00697=798156,1112951
EC00698=798156,1112951
EC00699=798156,1112951
EC00700=798156,1112951
EC00701=798156,1112951
EC00702=798156,1112951
EC00703=798156,1112951
EC00704=798156,1112951
EC00705=798156,1112951
EC00706=798156,1112951
EC00707=798156,1112951
EC00708=798156,1112951
EC00709=798156,1112951
EC00710=798156,1112951
EC00711=798156,1112951
EC00712=798156,1112951
EC00713=798156,1112951
EC00714=798156,1112951
EC00715=798156,1112951
EC00716=798156,1112951
EC00717=798156,1112951
EC00718=798156,1112951
EC00719=798156,1112951
EC00720=798156,1112951
EC00721=798156,1112951
EC00722=798156,1112951
EC00723=798156,1112951
EC00724=798156,1112951
EC00725=798156,1112951
EC00726=798156,1112951
EC00727=798156,1112951
EC00728=798156,1112951
EC00729=798156,1112951
EC00730=798156,1112951
EC00731=798156,1112951
EC00732=798156,1112951
EC00733=798156,1112951
EC00734=798156,1112951
EC00735=798156,1112951
EC00736=798156,1112951
EC00737=798156,1112951
EC00738=798156,1112951
EC00739=798156,1112951
EC00740=798156,1112951
EC00741=798156,1112951
EC00742=798156,1112951
EC00743=798156,1112951
EC00744=798156,1112951
EC00745=798156,1112951
EC00746=798156,1112951
EC00747=798156,1112951
EC00748=798156,1112951
EC00749=798156,1112951
EC00750=798156,1112951
EC00751=798156,1112951
EC00752=798156,1112951
EC00753=798156,1112951
EC00754=798156,1112951
///POSTYPE BASE
///RECTAN
///RCONF 0,0,0,0,0,0,0,0,0,0,0,0,0,0,0,0,0,0,0,0,0,0,0,0
P00006=0.222,-3.123,-1.508,0.0000,0.0000,0.0000
P00021=-0.225,-6.128,-0.405,0.0000,0.0000,0.0000
P00022=0.222,-3.123,-1.508,0.0000,0.0000,0.0000
P00023=0.143,-0.036,0.682,0.0000,0.0000,0.0000
P00024=0.145,-0.552,1.326,0.0000,0.0000,0.0000
P00025=-2.003,0.006,0.728,0.0000,0.0000,0.0000
P00026=0.562,-0.002,-0.337,0.0000,0.0000,0.0000
P00027=-0.746,0.015,-9.096,0.0000,0.0000,0.0000
P00028=-2.237,-0.018,-7.702,0.0000,0.0000,0.0000
P00029=-2.156,-0.086,-4.681,0.0000,0.0000,0.0000
P00030=5.926,-4.294,-1.390,0.0000,0.0000,0.0000
P00031=1.853,-0.001,-1.549,0.0000,0.0000,0.0000
P00032=1.957,0.503,-7.217,0.0000,0.0000,0.0000
///RCONF 0,0,0,0,1,0,0,0,0,0,0,0,0,0,0,0,0,0,0,0,0,0,0,0
P00033=-0.123,0.612,-5.012,0.0000,0.0000,0.0000
///RCONF 0,0,0,0,0,0,0,0,0,0,0,0,0,0,0,0,0,0,0,0,0,0,0,0
P00034=-0.304,0.773,-2.693,0.0000,0.0000,0.0000
P00042=-0.217,1.941,0.413,0.0000,0.0000,0.0000
P00043=-0.044,-1.937,1.197,0.0000,0.0000,0.0000
P00044=0.687,-2.322,1.156,0.0000,0.0000,0.0000
P00045=-0.068,-0.810,1.603,0.0000,0.0000,0.0000
P00046=0.799,0.043,1.292,0.0000,0.0000,0.0000
///RCONF 0,1,0,0,0,0,0,0,0,0,0,0,0,0,0,0,0,0,0,0,0,0,0,0
P00047=-0.011,1.737,-0.646,0.0000,0.0000,0.0000
///RCONF 0,0,0,0,0,0,0,0,0,0,0,0,0,0,0,0,0,0,0,0,0,0,0,0
P00048=2.411,0.025,-0.606,0.0000,0.0000,0.0000
P00049=3.413,-3.572,-1.618,0.0000,0.0000,0.0000
P00050=4.296,-4.501,-0.826,0.0000,0.0000,0.0000
P00051=0.367,3.892,0.009,0.0000,0.0000,0.0000
P00060=2.327,-2.514,-2.692,0.0000,0.0000,0.0000
//INST
///DATE 2025/03/12 10:01
///ATTR SC,RW
///GROUP1 RB1,BS1
///GROUP2 ST1
NOP
COMM 'X2_38-47,64(1)(90,180)
COMM 'Down
COMM MOVJ C00000 BC00000 VJ=100.00  +MOVJ EC00000 VJ=100.00
COMM 'Up
COMM 'Path S3659
COMM SFTOF3D
COMM MOVJ C00001 BC00001 VJ=100.00  +MOVJ EC00001 VJ=100.00
COMM MOVL C00002 BC00002 V=666.7  +MOVJ EC00002 VJ=100.00
COMM SMOVL C00003 BC00003 V=166.7  +MOVJ EC00003
COMM SREFP 3 C00004 BC00004  +REFP EC00004
COMM CALL JOB:SEARCH-R1-S13D
COMM SET P021 P006
COMM SFTON3D P021
COMM SMOVL C00005 BC00005 V=166.7  +MOVJ EC00005
COMM SREFP 3 C00006 BC00006  +REFP EC00006
COMM CALL JOB:SEARCH-R1-S13D
COMM SET P021 P006
COMM SFTON3D P021
COMM SMOVL C00007 BC00007 V=166.7  +MOVJ EC00007
COMM MOVL C00008 BC00008 V=1000.0  +MOVJ EC00008 VJ=100.00
COMM 'EndPath S3659
COMM 'Path S4334
COMM SFTOF3D
COMM MOVJ C00009 BC00009 VJ=100.00  +MOVJ EC00009 VJ=100.00
COMM MOVL C00010 BC00010 V=666.7  +MOVJ EC00010 VJ=100.00
COMM SMOVL C00011 BC00011 V=166.7  +MOVJ EC00011
COMM SREFP 3 C00012 BC00012  +REFP EC00012
COMM CALL JOB:SEARCH-R1-S13D
COMM SET P022 P006
COMM SFTON3D P022
COMM SMOVL C00013 BC00013 V=166.7  +MOVJ EC00013
COMM SREFP 3 C00014 BC00014  +REFP EC00014
COMM CALL JOB:SEARCH-R1-S13D
COMM SET P022 P006
COMM SFTON3D P022
COMM SMOVL C00015 BC00015 V=166.7  +MOVJ EC00015
COMM MOVL C00016 BC00016 V=1000.0  +MOVJ EC00016 VJ=100.00
COMM 'EndPath S4334
COMM 'Path S3657
COMM SFTOF3D
COMM MOVJ C00017 BC00017 VJ=100.00  +MOVJ EC00017 VJ=100.00
COMM MOVJ C00018 BC00018 VJ=100.00  +MOVJ EC00018 VJ=100.00
COMM MOVL C00019 BC00019 V=666.7  +MOVJ EC00019 VJ=100.00
COMM SMOVL C00020 BC00020 V=166.7  +MOVJ EC00020
COMM SREFP 3 C00021 BC00021  +REFP EC00021
COMM CALL JOB:SEARCH-R1-S13D
COMM SET P023 P006
COMM SFTON3D P023
COMM SMOVL C00022 BC00022 V=166.7  +MOVJ EC00022
COMM SREFP 3 C00023 BC00023  +REFP EC00023
COMM CALL JOB:SEARCH-R1-S13D
COMM SET P023 P006
COMM SFTON3D P023
COMM SMOVL C00024 BC00024 V=166.7  +MOVJ EC00024
COMM SMOVL C00025 BC00025 V=500.0  +MOVJ EC00025
COMM SMOVL C00026 BC00026 V=800.0  +MOVJ EC00026
COMM SMOVL C00027 BC00027 V=166.7  +MOVJ EC00027
COMM SREFP 3 C00028 BC00028  +REFP EC00028
COMM CALL JOB:SEARCH-R1-S13D
COMM SET P023 P006
COMM SFTON3D P023
COMM SMOVL C00029 BC00029 V=250.0  +MOVJ EC00029
COMM MOVL C00030 BC00030 V=1000.0  +MOVJ EC00030 VJ=100.00
COMM 'EndPath S3657
COMM MOVJ C00031 BC00031 VJ=100.00  +MOVJ EC00031 VJ=100.00
COMM 'Path S3665
COMM SFTOF3D
COMM MOVJ C00032 BC00032 VJ=100.00  +MOVJ EC00032 VJ=100.00
COMM MOVL C00033 BC00033 V=800.0  +MOVJ EC00033 VJ=100.00
COMM SMOVL C00034 BC00034 V=166.7  +MOVJ EC00034
COMM SREFP 3 C00035 BC00035  +REFP EC00035
COMM CALL JOB:SEARCH-R1-S13D
COMM SET P024 P006
COMM SFTON3D P024
COMM SMOVL C00036 BC00036 V=166.7  +MOVJ EC00036
COMM SMOVL C00037 BC00037 V=166.7  +MOVJ EC00037
COMM SREFP 3 C00038 BC00038  +REFP EC00038
COMM CALL JOB:SEARCH-R1-S13D
COMM SET P024 P006
COMM SFTON3D P024
COMM SMOVL C00039 BC00039 V=166.7  +MOVJ EC00039
COMM SMOVL C00040 BC00040 V=166.7  +MOVJ EC00040
COMM SREFP 3 C00041 BC00041  +REFP EC00041
COMM CALL JOB:SEARCH-R1-S13D
COMM SET P024 P006
COMM SFTON3D P024
COMM SMOVL C00042 BC00042 V=166.7  +MOVJ EC00042
COMM MOVL C00043 BC00043 V=1000.0  +MOVJ EC00043 VJ=100.00
COMM MOVL C00044 BC00044 V=1000.0  +MOVJ EC00044 VJ=100.00
COMM 'EndPath S3665
COMM 'Path S4335
COMM SFTOF3D
COMM MOVJ C00045 BC00045 VJ=100.00  +MOVJ EC00045 VJ=100.00
COMM MOVL C00046 BC00046 V=800.0  +MOVJ EC00046 VJ=100.00
COMM SMOVL C00047 BC00047 V=166.7  +MOVJ EC00047
COMM SREFP 3 C00048 BC00048  +REFP EC00048
COMM CALL JOB:SEARCH-R1-S13D
COMM SET P025 P006
COMM SFTON3D P025
COMM SMOVL C00049 BC00049 V=166.7  +MOVJ EC00049
COMM SMOVL C00050 BC00050 V=166.7  +MOVJ EC00050
COMM SREFP 3 C00051 BC00051  +REFP EC00051
COMM CALL JOB:SEARCH-R1-S13D
COMM SET P025 P006
COMM SFTON3D P025
COMM SMOVL C00052 BC00052 V=166.7  +MOVJ EC00052
COMM SMOVL C00053 BC00053 V=166.7  +MOVJ EC00053
COMM SREFP 3 C00054 BC00054  +REFP EC00054
COMM CALL JOB:SEARCH-R1-S13D
COMM SET P025 P006
COMM SFTON3D P025
COMM SMOVL C00055 BC00055 V=166.7  +MOVJ EC00055
COMM MOVL C00056 BC00056 V=1000.0  +MOVJ EC00056 VJ=100.00
COMM MOVL C00057 BC00057 V=1000.0  +MOVJ EC00057 VJ=100.00
COMM 'EndPath S4335
COMM 'Path S3666
COMM SFTOF3D
COMM MOVJ C00058 BC00058 VJ=100.00  +MOVJ EC00058 VJ=100.00
COMM MOVL C00059 BC00059 V=800.0  +MOVJ EC00059 VJ=100.00
COMM SMOVL C00060 BC00060 V=166.7  +MOVJ EC00060
COMM SREFP 3 C00061 BC00061  +REFP EC00061
COMM CALL JOB:SEARCH-R1-S13D
COMM SET P026 P006
COMM SFTON3D P026
COMM SMOVL C00062 BC00062 V=166.7  +MOVJ EC00062
COMM SREFP 3 C00063 BC00063  +REFP EC00063
COMM CALL JOB:SEARCH-R1-S13D
COMM SET P026 P006
COMM SFTON3D P026
COMM SMOVL C00064 BC00064 V=166.7  +MOVJ EC00064
COMM MOVL C00065 BC00065 V=1000.0  +MOVJ EC00065 VJ=100.00
COMM 'EndPath S3666
COMM MOVJ C00066 BC00066 VJ=100.00  +MOVJ EC00066 VJ=100.00
COMM MOVJ C00067 BC00067 VJ=100.00  +MOVJ EC00067 VJ=100.00
COMM 'Path S3661
COMM SFTOF3D
COMM MOVJ C00068 BC00068 VJ=100.00  +MOVJ EC00068 VJ=100.00
COMM MOVL C00069 BC00069 V=800.0  +MOVJ EC00069 VJ=100.00
COMM SMOVL C00070 BC00070 V=166.7  +MOVJ EC00070
COMM SREFP 3 C00071 BC00071  +REFP EC00071
COMM CALL JOB:SEARCH-R1-S13D
COMM SET P027 P006
COMM SFTON3D P027
COMM SMOVL C00072 BC00072 V=166.7  +MOVJ EC00072
COMM SMOVL C00073 BC00073 V=166.7  +MOVJ EC00073
COMM SREFP 3 C00074 BC00074  +REFP EC00074
COMM CALL JOB:SEARCH-R1-S13D
COMM SET P027 P006
COMM SFTON3D P027
COMM SMOVL C00075 BC00075 V=250.0  +MOVJ EC00075
COMM SMOVL C00076 BC00076 V=166.7  +MOVJ EC00076
COMM SREFP 3 C00077 BC00077  +REFP EC00077
COMM CALL JOB:SEARCH-R1-S13D
COMM SET P027 P006
COMM SFTON3D P027
COMM SMOVL C00078 BC00078 V=166.7  +MOVJ EC00078
COMM MOVL C00079 BC00079 V=1000.0  +MOVJ EC00079 VJ=100.00
COMM MOVL C00080 BC00080 V=1000.0  +MOVJ EC00080 VJ=100.00
COMM 'EndPath S3661
COMM 'Path S4336
COMM SFTOF3D
COMM MOVJ C00081 BC00081 VJ=100.00  +MOVJ EC00081 VJ=100.00
COMM MOVL C00082 BC00082 V=800.0  +MOVJ EC00082 VJ=100.00
COMM SMOVL C00083 BC00083 V=166.7  +MOVJ EC00083
COMM SREFP 3 C00084 BC00084  +REFP EC00084
COMM CALL JOB:SEARCH-R1-S13D
COMM SET P028 P006
COMM SFTON3D P028
COMM SMOVL C00085 BC00085 V=166.7  +MOVJ EC00085
COMM SREFP 3 C00086 BC00086  +REFP EC00086
COMM CALL JOB:SEARCH-R1-S13D
COMM SET P028 P006
COMM SFTON3D P028
COMM SMOVL C00087 BC00087 V=166.7  +MOVJ EC00087
COMM MOVL C00088 BC00088 V=1000.0  +MOVJ EC00088 VJ=100.00
COMM 'EndPath S4336
COMM MOVJ C00089 BC00089 VJ=100.00  +MOVJ EC00089 VJ=100.00
COMM 'Path S4879
COMM SFTOF3D
COMM MOVJ C00090 BC00090 VJ=100.00  +MOVJ EC00090 VJ=100.00
COMM MOVL C00091 BC00091 V=800.0  +MOVJ EC00091 VJ=100.00
COMM SMOVL C00092 BC00092 V=166.7  +MOVJ EC00092
COMM SREFP 3 C00093 BC00093  +REFP EC00093
COMM CALL JOB:SEARCH-R1-S13D
COMM SET P060 P006
COMM SFTON3D P060
COMM SMOVL C00094 BC00094 V=166.7  +MOVJ EC00094
COMM SMOVL C00095 BC00095 V=166.7  +MOVJ EC00095
COMM SREFP 3 C00096 BC00096  +REFP EC00096
COMM CALL JOB:SEARCH-R1-S13D
COMM SET P060 P006
COMM SFTON3D P060
COMM SMOVL C00097 BC00097 V=166.7  +MOVJ EC00097
COMM SMOVL C00098 BC00098 V=250.0  +MOVJ EC00098
COMM SMOVL C00099 BC00099 V=166.7  +MOVJ EC00099
COMM SREFP 3 C00100 BC00100  +REFP EC00100
COMM CALL JOB:SEARCH-R1-S13D
COMM SET P060 P006
COMM SFTON3D P060
COMM SMOVL C00101 BC00101 V=166.7  +MOVJ EC00101
COMM MOVL C00102 BC00102 V=1000.0  +MOVJ EC00102 VJ=100.00
COMM 'EndPath S4879
COMM MOVJ C00103 BC00103 VJ=100.00  +MOVJ EC00103 VJ=100.00
COMM 'Path S3664
COMM SFTOF3D
COMM MOVJ C00104 BC00104 VJ=100.00  +MOVJ EC00104 VJ=100.00
COMM MOVL C00105 BC00105 V=800.0  +MOVJ EC00105 VJ=100.00
COMM SMOVL C00106 BC00106 V=166.7  +MOVJ EC00106
COMM SREFP 3 C00107 BC00107  +REFP EC00107
COMM CALL JOB:SEARCH-R1-S13D
COMM SET P029 P006
COMM SFTON3D P029
COMM SMOVL C00108 BC00108 V=166.7  +MOVJ EC00108
COMM SREFP 3 C00109 BC00109  +REFP EC00109
COMM CALL JOB:SEARCH-R1-S13D
COMM SET P029 P006
COMM SFTON3D P029
COMM SMOVL C00110 BC00110 V=166.7  +MOVJ EC00110
COMM MOVL C00111 BC00111 V=1000.0  +MOVJ EC00111 VJ=100.00
COMM 'EndPath S3664
COMM 'Path S4337
COMM SFTOF3D
COMM MOVJ C00112 BC00112 VJ=100.00  +MOVJ EC00112 VJ=100.00
COMM MOVL C00113 BC00113 V=800.0  +MOVJ EC00113 VJ=100.00
COMM SMOVL C00114 BC00114 V=166.7  +MOVJ EC00114
COMM SREFP 3 C00115 BC00115  +REFP EC00115
COMM CALL JOB:SEARCH-R1-S13D
COMM SET P030 P006
COMM SFTON3D P030
COMM SMOVL C00116 BC00116 V=166.7  +MOVJ EC00116
COMM SREFP 3 C00117 BC00117  +REFP EC00117
COMM CALL JOB:SEARCH-R1-S13D
COMM SET P030 P006
COMM SFTON3D P030
COMM SMOVL C00118 BC00118 V=166.7  +MOVJ EC00118
COMM MOVL C00119 BC00119 V=800.0  +MOVJ EC00119 VJ=100.00
COMM MOVL C00120 BC00120 V=1000.0  +MOVJ EC00120 VJ=100.00
COMM 'EndPath S4337
COMM MOVJ C00121 BC00121 VJ=100.00  +MOVJ EC00121 VJ=100.00
COMM 'Path S3663
COMM SFTOF3D
COMM MOVJ C00122 BC00122 VJ=100.00  +MOVJ EC00122 VJ=100.00
COMM MOVL C00123 BC00123 V=800.0  +MOVJ EC00123 VJ=100.00
COMM SMOVL C00124 BC00124 V=166.7  +MOVJ EC00124
COMM SREFP 3 C00125 BC00125  +REFP EC00125
COMM CALL JOB:SEARCH-R1-S13D
COMM SET P031 P006
COMM SFTON3D P031
COMM SMOVL C00126 BC00126 V=166.7  +MOVJ EC00126
COMM SREFP 3 C00127 BC00127  +REFP EC00127
COMM CALL JOB:SEARCH-R1-S13D
COMM SET P031 P006
COMM SFTON3D P031
COMM SMOVL C00128 BC00128 V=166.7  +MOVJ EC00128
COMM SMOVL C00129 BC00129 V=166.7  +MOVJ EC00129
COMM SREFP 3 C00130 BC00130  +REFP EC00130
COMM CALL JOB:SEARCH-R1-S13D
COMM SET P031 P006
COMM SFTON3D P031
COMM SMOVL C00131 BC00131 V=166.7  +MOVJ EC00131
COMM MOVL C00132 BC00132 V=1000.0  +MOVJ EC00132 VJ=100.00
COMM 'EndPath S3663
COMM MOVJ C00133 BC00133 VJ=100.00  +MOVJ EC00133 VJ=100.00
COMM 'Path S4338
COMM SFTOF3D
COMM MOVJ C00134 BC00134 VJ=100.00  +MOVJ EC00134 VJ=100.00
COMM MOVL C00135 BC00135 V=800.0  +MOVJ EC00135 VJ=100.00
COMM SMOVL C00136 BC00136 V=166.7  +MOVJ EC00136
COMM SREFP 3 C00137 BC00137  +REFP EC00137
COMM CALL JOB:SEARCH-R1-S13D
COMM SET P032 P006
COMM SFTON3D P032
COMM SMOVL C00138 BC00138 V=166.7  +MOVJ EC00138
COMM SREFP 3 C00139 BC00139  +REFP EC00139
COMM CALL JOB:SEARCH-R1-S13D
COMM SET P032 P006
COMM SFTON3D P032
COMM SMOVL C00140 BC00140 V=166.7  +MOVJ EC00140
COMM SMOVL C00141 BC00141 V=166.7  +MOVJ EC00141
COMM SREFP 3 C00142 BC00142  +REFP EC00142
COMM CALL JOB:SEARCH-R1-S13D
COMM SET P032 P006
COMM SFTON3D P032
COMM SMOVL C00143 BC00143 V=166.7  +MOVJ EC00143
COMM MOVL C00144 BC00144 V=1000.0  +MOVJ EC00144 VJ=100.00
COMM 'EndPath S4338
COMM MOVJ C00145 BC00145 VJ=100.00  +MOVJ EC00145 VJ=100.00
COMM 'Path S3662
COMM SFTOF3D
COMM MOVJ C00146 BC00146 VJ=100.00  +MOVJ EC00146 VJ=100.00
COMM MOVL C00147 BC00147 V=800.0  +MOVJ EC00147 VJ=100.00
COMM SMOVL C00148 BC00148 V=166.7  +MOVJ EC00148
COMM SREFP 3 C00149 BC00149  +REFP EC00149
COMM CALL JOB:SEARCH-R1-S13D
COMM SET P033 P006
COMM SFTON3D P033
COMM SMOVL C00150 BC00150 V=166.7  +MOVJ EC00150
COMM SREFP 3 C00151 BC00151  +REFP EC00151
COMM CALL JOB:SEARCH-R1-S13D
COMM SET P033 P006
COMM SFTON3D P033
COMM SMOVL C00152 BC00152 V=166.7  +MOVJ EC00152
COMM MOVL C00153 BC00153 V=1000.0  +MOVJ EC00153 VJ=100.00
COMM 'EndPath S3662
COMM 'Path S4339
COMM SFTOF3D
COMM MOVJ C00154 BC00154 VJ=100.00  +MOVJ EC00154 VJ=100.00
COMM MOVL C00155 BC00155 V=800.0  +MOVJ EC00155 VJ=100.00
COMM SMOVL C00156 BC00156 V=166.7  +MOVJ EC00156
COMM SREFP 3 C00157 BC00157  +REFP EC00157
COMM CALL JOB:SEARCH-R1-S13D
COMM SET P034 P006
COMM SFTON3D P034
COMM SMOVL C00158 BC00158 V=166.7  +MOVJ EC00158
COMM SMOVL C00159 BC00159 V=166.7  +MOVJ EC00159
COMM SREFP 3 C00160 BC00160  +REFP EC00160
COMM CALL JOB:SEARCH-R1-S13D
COMM SET P034 P006
COMM SFTON3D P034
COMM SMOVL C00161 BC00161 V=166.7  +MOVJ EC00161
COMM SMOVL C00162 BC00162 V=166.7  +MOVJ EC00162
COMM SREFP 3 C00163 BC00163  +REFP EC00163
COMM CALL JOB:SEARCH-R1-S13D
COMM SET P034 P006
COMM SFTON3D P034
COMM SMOVL C00164 BC00164 V=166.7  +MOVJ EC00164
COMM MOVL C00165 BC00165 V=1000.0  +MOVJ EC00165 VJ=100.00
COMM 'EndPath S4339
COMM MOVJ C00166 BC00166 VJ=100.00  +MOVJ EC00166 VJ=100.00
COMM 'Path W3667
COMM SFTOF3D
COMM SFTON3D P026
COMM MOVJ C00167 BC00167 VJ=100.00  +MOVJ EC00167 VJ=100.00
COMM SMOVL C00168 BC00168 V=800.0  +MOVJ EC00168
COMM SREFP 1 C00169 BC00169  +REFP EC00169
COMM SREFP 2 C00170 BC00170  +REFP EC00170
COMM SMOVL C00171 BC00171 V=166.7 PL=0  +MOVJ EC00171
COMM MACRO1 MJ#(0) ARGF21
COMM ARCON
COMM SWVON WEV#(100)
COMM SMOVL C00172 BC00172 V=9.2  +MOVJ EC00172
COMM SMOVL C00173 BC00173 V=9.2  +MOVJ EC00173
COMM SMOVL C00174 BC00174 V=9.2  +MOVJ EC00174
COMM ARCOF
COMM SWVOF
COMM SMOVL C00175 BC00175 V=800.0  +MOVJ EC00175
COMM SMOVL C00176 BC00176 V=1000.0  +MOVJ EC00176
COMM SFTOF3D
COMM 'EndPath W3667
COMM MOVJ C00177 BC00177 VJ=100.00  +MOVJ EC00177 VJ=100.00
COMM MOVJ C00178 BC00178 VJ=100.00  +MOVJ EC00178 VJ=100.00
COMM 'Path W3668
COMM SSFTOF
COMM SFTOF3D
COMM SFTON3D P028
COMM MOVJ C00179 BC00179 VJ=100.00  +MOVJ EC00179 VJ=100.00
COMM SMOVL C00180 BC00180 V=800.0  +MOVJ EC00180
COMM SREFP 1 C00181 BC00181  +REFP EC00181
COMM SREFP 2 C00182 BC00182  +REFP EC00182
COMM SMOVL C00183 BC00183 V=150.0 PL=0  +MOVJ EC00183
COMM ARCON
COMM SWVON WEV#(100)
COMM SFTON3D P027
COMM SMOVL C00184 BC00184 V=9.2  +MOVJ EC00184
COMM SMOVL C00185 BC00185 V=9.2  +MOVJ EC00185
COMM ARCOF
COMM SWVOF
COMM SMOVL C00186 BC00186 V=800.0  +MOVJ EC00186
COMM SMOVL C00187 BC00187 V=1000.0  +MOVJ EC00187
COMM SFTOF3D
COMM 'EndPath W3668
COMM MOVJ C00188 BC00188 VJ=100.00  +MOVJ EC00188 VJ=100.00
COMM 'Path W4546
COMM SFTOF3D
COMM SFTON3D P022
COMM MOVJ C00189 BC00189 VJ=100.00  +MOVJ EC00189 VJ=100.00
COMM SMOVL C00190 BC00190 V=800.0  +MOVJ EC00190
COMM SMOVL C00191 BC00191 V=150.0 PL=0  +MOVJ EC00191
COMM MACRO1 MJ#(0) ARGF9
COMM ARCON
COMM SWVON WEV#(10)
COMM SFTON3D P021
COMM SMOVL C00192 BC00192 V=10.0  +MOVJ EC00192
COMM ARCOF
COMM SWVOF
COMM SMOVL C00193 BC00193 V=800.0  +MOVJ EC00193
COMM SMOVL C00194 BC00194 V=1000.0  +MOVJ EC00194
COMM SFTOF3D
COMM 'EndPath W4546
COMM 'Path W4901
COMM SFTOF3D
COMM SFTON3D P060
COMM MOVJ C00195 BC00195 VJ=100.00  +MOVJ EC00195 VJ=100.00
COMM MOVJ C00196 BC00196 VJ=100.00  +MOVJ EC00196 VJ=100.00
COMM MOVJ C00197 BC00197 VJ=100.00  +MOVJ EC00197 VJ=100.00
COMM SMOVL C00198 BC00198 V=800.0  +MOVJ EC00198
COMM SMOVL C00199 BC00199 V=150.0 PL=0  +MOVJ EC00199
COMM MACRO1 MJ#(0) ARGF14
COMM ARCON
COMM SMOVL C00200 BC00200 V=10.8  +MOVJ EC00200
COMM ARCOF
COMM SMOVL C00201 BC00201 V=800.0  +MOVJ EC00201
COMM SFTOF3D
COMM 'EndPath W4901
COMM 'Path W4880
COMM SFTOF3D
COMM SFTON3D P060
COMM SMOVL C00202 BC00202 V=800.0  +MOVJ EC00202
COMM SMOVL C00203 BC00203 V=150.0 PL=0  +MOVJ EC00203
COMM ARCON
COMM SMOVL C00204 BC00204 V=10.0  +MOVJ EC00204
COMM SMOVL C00205 BC00205 V=10.0  +MOVJ EC00205
COMM SMOVL C00206 BC00206 V=10.0  +MOVJ EC00206
COMM ARCOF
COMM SMOVL C00207 BC00207 V=800.0  +MOVJ EC00207
COMM SMOVL C00208 BC00208 V=1000.0  +MOVJ EC00208
COMM SFTOF3D
COMM 'EndPath W4880
COMM MOVJ C00209 BC00209 VJ=100.00  +MOVJ EC00209 VJ=100.00
COMM MOVJ C00210 BC00210 VJ=100.00  +MOVJ EC00210 VJ=100.00
COMM 'Path W4548
COMM SFTOF3D
COMM SFTON3D P030
COMM MOVJ C00211 BC00211 VJ=100.00  +MOVJ EC00211 VJ=100.00
COMM SMOVL C00212 BC00212 V=800.0  +MOVJ EC00212
COMM SMOVL C00213 BC00213 V=150.0 PL=0  +MOVJ EC00213
COMM MACRO1 MJ#(0) ARGF9
COMM ARCON
COMM SFTON3D P029
COMM SMOVL C00214 BC00214 V=10.0  +MOVJ EC00214
COMM SMOVL C00215 BC00215 V=10.0  +MOVJ EC00215
COMM ARCOF
COMM SMOVL C00216 BC00216 V=800.0  +MOVJ EC00216
COMM SMOVL C00217 BC00217 V=1000.0  +MOVJ EC00217
COMM SFTOF3D
COMM 'EndPath W4548
COMM MOVJ C00218 BC00218 VJ=100.00  +MOVJ EC00218 VJ=100.00
COMM MOVJ C00219 BC00219 VJ=100.00  +MOVJ EC00219 VJ=100.00
COMM 'Path W3671
COMM SFTOF3D
COMM SFTON3D P033
COMM MOVJ C00220 BC00220 VJ=100.00  +MOVJ EC00220 VJ=100.00
COMM SMOVL C00221 BC00221 V=800.0  +MOVJ EC00221
COMM SMOVL C00222 BC00222 V=166.7 PL=0  +MOVJ EC00222
COMM MACRO1 MJ#(0) ARGF14
COMM ARCON
COMM SMOVL C00223 BC00223 V=9.2  +MOVJ EC00223
COMM SFTON3D P034
COMM SMOVL C00224 BC00224 V=9.2  +MOVJ EC00224
COMM SMOVL C00225 BC00225 V=9.2  +MOVJ EC00225
COMM ARCOF
COMM SMOVL C00226 BC00226 V=800.0  +MOVJ EC00226
COMM SMOVL C00227 BC00227 V=1000.0  +MOVJ EC00227
COMM SFTOF3D
COMM 'EndPath W3671
COMM MOVJ C00228 BC00228 VJ=100.00  +MOVJ EC00228 VJ=100.00
COMM 'Path W3672
COMM SFTOF3D
COMM SFTON3D P024
COMM MOVJ C00229 BC00229 VJ=100.00  +MOVJ EC00229 VJ=100.00
COMM SMOVL C00230 BC00230 V=800.0  +MOVJ EC00230
COMM SMOVL C00231 BC00231 V=166.7 PL=0  +MOVJ EC00231
COMM ARCON
COMM SMOVL C00232 BC00232 V=9.2  +MOVJ EC00232
COMM SFTON3D P025
COMM SMOVL C00233 BC00233 V=9.2  +MOVJ EC00233
COMM SMOVL C00234 BC00234 V=9.2  +MOVJ EC00234
COMM ARCOF
COMM SMOVL C00235 BC00235 V=800.0  +MOVJ EC00235
COMM SMOVL C00236 BC00236 V=1000.0  +MOVJ EC00236
COMM SFTOF3D
COMM 'EndPath W3672
COMM MOVJ C00237 BC00237 VJ=100.00  +MOVJ EC00237 VJ=100.00
COMM 'Path W3673
COMM SFTOF3D
COMM SFTON3D P032
COMM MOVJ C00238 BC00238 VJ=100.00  +MOVJ EC00238 VJ=100.00
COMM SMOVL C00239 BC00239 V=800.0  +MOVJ EC00239
COMM SMOVL C00240 BC00240 V=166.7 PL=0  +MOVJ EC00240
COMM ARCON
COMM SMOVL C00241 BC00241 V=9.2  +MOVJ EC00241
COMM SFTON3D P031
COMM SMOVL C00242 BC00242 V=9.2  +MOVJ EC00242
COMM SMOVL C00243 BC00243 V=9.2  +MOVJ EC00243
COMM ARCOF
COMM SMOVL C00244 BC00244 V=800.0  +MOVJ EC00244
COMM SMOVL C00245 BC00245 V=1000.0  +MOVJ EC00245
COMM SFTOF3D
COMM 'EndPath W3673
COMM MOVJ C00246 BC00246 VJ=100.00  +MOVJ EC00246 VJ=100.00
COMM '
COMM MOVJ C00247 BC00247 VJ=100.00  +MOVJ EC00247 VJ=100.00
COMM JUMP *VV
COMM MOVJ C00248 BC00248 VJ=100.00  +MOVJ EC00248 VJ=100.00
COMM 'Path W3680
COMM SFTOF3D
COMM SFTON3D P023
COMM MOVJ C00249 BC00249 VJ=100.00  +MOVJ EC00249 VJ=100.00
COMM SMOVL C00250 BC00250 V=800.0  +MOVJ EC00250
COMM SMOVL C00251 BC00251 V=166.7 PL=0  +MOVJ EC00251
COMM SMOVL C00252 BC00252 V=10.0  +MOVJ EC00252
COMM SMOVL C00253 BC00253 V=33.3  +MOVJ EC00253
COMM SMOVL C00254 BC00254 V=33.3  +MOVJ EC00254
COMM SMOVL C00255 BC00255 V=33.3  +MOVJ EC00255
COMM SMOVL C00256 BC00256 V=10.0  +MOVJ EC00256
COMM SMOVL C00257 BC00257 V=10.0  +MOVJ EC00257
COMM SMOVL C00258 BC00258 V=10.0  +MOVJ EC00258
COMM SMOVL C00259 BC00259 V=10.0  +MOVJ EC00259
COMM SMOVL C00260 BC00260 V=10.0  +MOVJ EC00260
COMM ARCOF
COMM SMOVL C00261 BC00261 V=800.0  +MOVJ EC00261
COMM SMOVL C00262 BC00262 V=1000.0  +MOVJ EC00262
COMM SFTOF3D
COMM 'EndPath W3680
COMM 'Path W3681
COMM *VV
COMM SFTOF3D
COMM SFTON3D P023
COMM MOVJ C00263 BC00263 VJ=100.00  +MOVJ EC00263 VJ=100.00
COMM SMOVL C00264 BC00264 V=800.0  +MOVJ EC00264
COMM SMOVL C00265 BC00265 V=150.0 PL=0  +MOVJ EC00265
COMM MACRO1 MJ#(0) ARGF9
COMM ARCON
COMM SMOVL C00266 BC00266 V=8.3  +MOVJ EC00266
COMM SMOVL C00267 BC00267 V=8.3  +MOVJ EC00267
COMM SMOVL C00268 BC00268 V=8.3  +MOVJ EC00268
COMM SMOVL C00269 BC00269 V=8.3  +MOVJ EC00269
COMM SMOVL C00270 BC00270 V=8.3  +MOVJ EC00270
COMM SMOVL C00271 BC00271 V=8.3  +MOVJ EC00271
COMM SMOVL C00272 BC00272 V=8.3  +MOVJ EC00272
COMM SMOVL C00273 BC00273 V=8.3  +MOVJ EC00273
COMM SMOVL C00274 BC00274 V=8.3  +MOVJ EC00274
COMM ARCOF
COMM SMOVL C00275 BC00275 V=800.0  +MOVJ EC00275
COMM SMOVL C00276 BC00276 V=1000.0  +MOVJ EC00276
COMM SFTOF3D
COMM 'EndPath W3681
COMM 'Down
COMM MOVJ C00277 BC00277 VJ=100.00  +MOVJ EC00277 VJ=100.00
COMM CALL JOB:CLEAN-R1_KM_NEW
'X2_38-47,64(1)(90,180)
'Down
MOVJ C00278 BC00278 VJ=100.00  +MOVJ EC00278 VJ=100.00
'Up
'Path S3659
SFTOF3D
MOVJ C00279 BC00279 VJ=100.00  +MOVJ EC00279 VJ=100.00
COMM PAUSE
COMM MOVL C00280 BC00280 V=666.7  +MOVJ EC00280 VJ=100.00
COMM SMOVL C00281 BC00281 V=166.7  +MOVJ EC00281
COMM SREFP 3 C00282 BC00282  +REFP EC00282
COMM CALL JOB:SEARCH-R1-S13D
COMM SET P021 P006
COMM SFTON3D P021
COMM SMOVL C00283 BC00283 V=166.7  +MOVJ EC00283
COMM SREFP 3 C00284 BC00284  +REFP EC00284
COMM CALL JOB:SEARCH-R1-S13D
COMM SET P021 P006
COMM SFTON3D P021
COMM SMOVL C00285 BC00285 V=166.7  +MOVJ EC00285
COMM MOVL C00286 BC00286 V=1000.0  +MOVJ EC00286 VJ=100.00
COMM 'EndPath S3659
COMM 'Path S4334
COMM SFTOF3D
COMM MOVJ C00287 BC00287 VJ=100.00  +MOVJ EC00287 VJ=100.00
COMM MOVL C00288 BC00288 V=666.7  +MOVJ EC00288 VJ=100.00
COMM SMOVL C00289 BC00289 V=166.7  +MOVJ EC00289
COMM SREFP 3 C00290 BC00290  +REFP EC00290
COMM CALL JOB:SEARCH-R1-S13D
COMM SET P022 P006
COMM SFTON3D P022
COMM SMOVL C00291 BC00291 V=166.7  +MOVJ EC00291
COMM SREFP 3 C00292 BC00292  +REFP EC00292
COMM CALL JOB:SEARCH-R1-S13D
COMM SET P022 P006
COMM SFTON3D P022
COMM SMOVL C00293 BC00293 V=166.7  +MOVJ EC00293
COMM MOVL C00294 BC00294 V=1000.0  +MOVJ EC00294 VJ=100.00
COMM 'EndPath S4334
COMM 'Path S3657
SFTOF3D
MOVJ C00295 BC00295 VJ=100.00  +MOVJ EC00295 VJ=100.00
MOVJ C00296 BC00296 VJ=100.00  +MOVJ EC00296 VJ=100.00
MOVL C00297 BC00297 V=666.7  +MOVJ EC00297 VJ=100.00
SMOVL C00298 BC00298 V=166.7  +MOVJ EC00298
SREFP 3 C00299 BC00299  +REFP EC00299
CALL JOB:SEARCH-R1-S13D
SET P023 P006
SFTON3D P023
SMOVL C00300 BC00300 V=166.7  +MOVJ EC00300
SREFP 3 C00301 BC00301  +REFP EC00301
CALL JOB:SEARCH-R1-S13D
SET P023 P006
SFTON3D P023
SMOVL C00302 BC00302 V=166.7  +MOVJ EC00302
SMOVL C00303 BC00303 V=500.0  +MOVJ EC00303
SMOVL C00304 BC00304 V=800.0  +MOVJ EC00304
SMOVL C00305 BC00305 V=166.7  +MOVJ EC00305
SREFP 3 C00306 BC00306  +REFP EC00306
CALL JOB:SEARCH-R1-S13D
SET P023 P006
SFTON3D P023
SMOVL C00307 BC00307 V=250.0  +MOVJ EC00307
MOVL C00308 BC00308 V=1000.0  +MOVJ EC00308 VJ=100.00
'EndPath S3657
MOVJ C00309 BC00309 VJ=100.00  +MOVJ EC00309 VJ=100.00
'Path S3665
SFTOF3D
MOVJ C00310 BC00310 VJ=100.00  +MOVJ EC00310 VJ=100.00
MOVL C00311 BC00311 V=800.0  +MOVJ EC00311 VJ=100.00
SMOVL C00312 BC00312 V=166.7  +MOVJ EC00312
SREFP 3 C00313 BC00313  +REFP EC00313
CALL JOB:SEARCH-R1-S13D
SET P024 P006
SFTON3D P024
